(* Logix 5000 project; controller BTS01 vendor 1 type 14 code 217 rev 32.14; software revision 32.04; part 2 of 15 *)
(* tags used below, declared in another part *)
   V1101 : DTE_Air_Valve_v2;   // Tank 1100 Fill Valve
   V1102 : DTE_Air_Valve_v2;   // Tank 1100 Discharge Valve
   V1103 : DTE_Air_Valve_v2;   // Tank 1100 Line Valve
   V1201 : DTE_Air_Valve_v2;   // Tank 1200 Fill Valve
   V1202 : DTE_Air_Valve_v2;   // Tank 1200 Discharge Valve
   V1203 : DTE_Air_Valve_v2;   // Tank 1200 Line Valve

ADD_ON_INSTRUCTION SCP   (* revision 1.2, vendor Rockwell Automation *)
// Scale w/Parameters
// Help:
// Use this instruction to scale data from your analog module and bring it into the limits prescribed by the process variable or another analog module.
// Equations used in calculating a linear relationship:
// Scaled value = (input value - input min.) x rate + scaled minimum
// Rate = (scaled max. - scaled min.) / (input max. - input min.)
// Enabling the Limit_En Bit Limits the Output Value to the Scaled Min/Max Values. (09/16/16) DTK
VAR_INPUT
   Input : REAL; {required}
   Input_Min : REAL; {required}
   Input_Max : REAL; {required}
   Scaled_Min : REAL; {required}
   Scaled_Max : REAL; {required}
END_VAR
VAR_OUTPUT
   Output : REAL; {access Read Only, required}
END_VAR
VAR_INPUT
   Limit_En : BOOL; {visible}   // Limit Enable Bit Limits Output to Scaled Min/Max Values
END_VAR
VAR
   Rate : REAL;
END_VAR

ROUTINE Logic   (* ladder *)
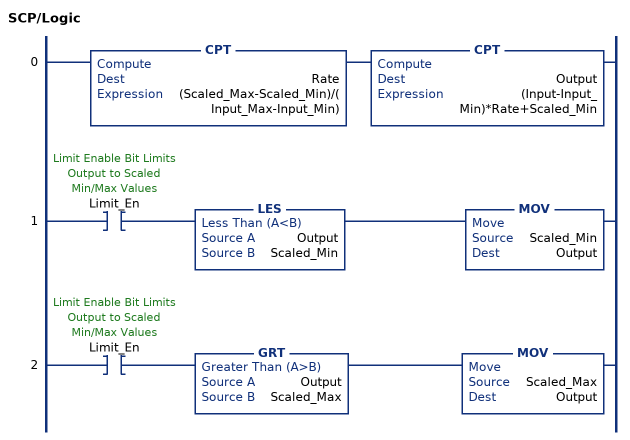
   0: CPT(Rate,(Scaled_Max-Scaled_Min)/(Input_Max-Input_Min))CPT(Output,(Input-Input_Min)*Rate+Scaled_Min);
   1: XIC(Limit_En)LES(Output,Scaled_Min)MOV(Scaled_Min,Output);
   2: XIC(Limit_En)GRT(Output,Scaled_Max)MOV(Scaled_Max,Output);
END_ROUTINE
END_ADD_ON_INSTRUCTION

ADD_ON_INSTRUCTION Temperature_Transmitter   (* revision 1.0 *)
VAR_INPUT
   RawInput : REAL; {required}   // Raw Input from Analog Input Card
   Input_Min : REAL; {required}   // I/O Module Scaling (MIN)
   Input_Max : REAL; {required}   // I/O Module Scaling (MAX)
   ScaledMin : REAL; {required}   // R/I Scaling (MIN)
   ScaledMax : REAL; {required}   // R/I Scaling (MAX)
   CalOffset : REAL; {required}   // Calibration Offset
END_VAR
VAR_OUTPUT
   MeasuredDegC : REAL; {access Read Only, visible}   // Sensor Temperature in Degrees C
   DegC : REAL; {access Read Only, visible}   // Display Temperature in Degrees C
   DegF : REAL; {access Read Only, visible}   // Display Temperature in Degrees F
END_VAR
VAR
   Offset : REAL;   // Linearity Offset
   Slope : REAL;   // Linearity Slope
END_VAR

ROUTINE Logic   (* ladder *)
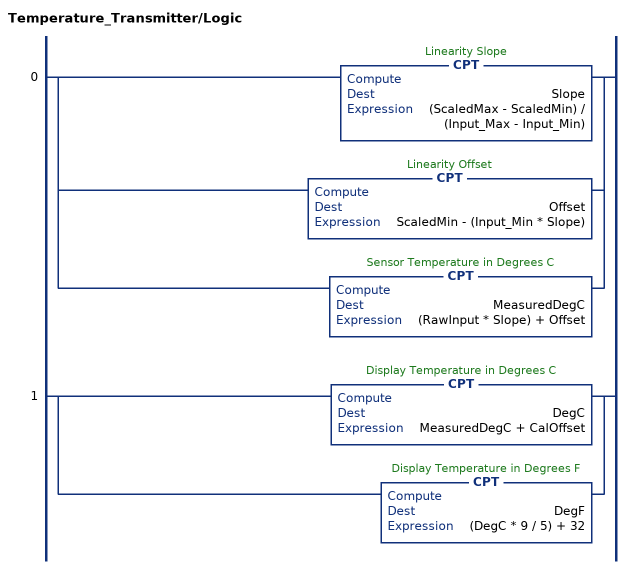
   0: [CPT(Slope,(ScaledMax - ScaledMin) / (Input_Max - Input_Min)) ,CPT(Offset,ScaledMin - (Input_Min * Slope)) ,CPT(MeasuredDegC,(RawInput * Slope) + Offset) ];
   1: [CPT(DegC,MeasuredDegC + CalOffset) ,CPT(DegF,(DegC * 9 / 5) + 32) ];
END_ROUTINE
END_ADD_ON_INSTRUCTION

ADD_ON_INSTRUCTION Toggle_Bit   (* revision 1.0 Created 4/01/2022 Sean Daehn *)
// Toggle Bit on and off with single momentary pushbutton
VAR_INPUT
   Toggle_PB : BOOL; {access None, required}
END_VAR
VAR_OUTPUT
   Output : BOOL; {access None, required}
END_VAR
VAR
   oneshot : BOOL; {access None}
   Toggle_On : BOOL; {access None}
   Toggle_Off : BOOL; {access None}
END_VAR

ROUTINE Logic   (* ladder *)
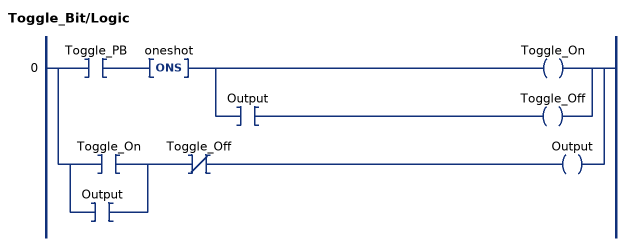
   0: [XIC(Toggle_PB) ONS(oneshot) [OTE(Toggle_On) ,XIC(Output) OTE(Toggle_Off) ] ,[XIC(Toggle_On) ,XIC(Output) ] XIO(Toggle_Off) OTE(Output) ];
END_ROUTINE
END_ADD_ON_INSTRUCTION

VAR_GLOBAL   (* controller tags *)
   ActiveRecipePF1000Interlock : DINT;
   AG1101 : DTE_VFD := (INTERLOCK := 1, SPEED_FWD := 20.0, AUTO_SPEED_SETPOINT := 20.0, FORCE_SPEED_SETPOINT := 10.0, ITEMTAG := 1101, MOA_MODE := 1);   // Tank 1100 Agitator
   AG1101_CIP_ENABLE : BOOL;
   AG1101_ONS : DINT := 1;
   AG1201 : DTE_VFD := (INTERLOCK := 1, SPEED_FWD := 20.0, AUTO_SPEED_SETPOINT := 20.0, FORCE_SPEED_SETPOINT := 20.0, ITEMTAG := 1201, MOA_MODE := 1);   // Tank 1200 Agitator
   AG1201_CIP_ENABLE : BOOL;
   AG1201_ONS : DINT;
   AirBlow_ONS : DINT;
   AirBlow_Timer : TIMER := (PRE := 30000);
   AirblowPB : BOOL;
   Alarm_Active : DINT;
   Alarm_TMR : TIMER[17,32] := ([0,0].PRE := 500, [0,1].PRE := 500, [0,2].PRE := 500, [0,3].PRE := 500, [0,4].PRE := 500, [0,5].PRE := 500, [0,6].PRE := 500, [0,7].PRE := 500, [0,8].PRE := 500, [0,9].PRE := 500, [0,10].PRE := 500, [0,11].PRE := 500, [0,12].PRE := 500, [0,13].PRE := 500, [0,14].PRE := 500, [0,15].PRE := 500, [0,16].PRE := 500, [0,17].PRE := 500, [0,18].PRE := 500, [0,19].PRE := 500, [0,20].PRE := 500, [0,21].PRE := 100, [0,22].PRE := 100, [0,23].PRE := 5000, [0,24].PRE := 5000, [0,25].PRE := 5000, [0,26].PRE := 5000, [0,27].PRE := 5000, [0,28].PRE := 5000, [0,29].PRE := 5000, [0,30].PRE := 5000, [0,31].PRE := 5000, [1,0].PRE := 100, [1,1].PRE := 100, [1,2].PRE := 500, [1,3].PRE := 500, [1,4].PRE := 500, [1,5].PRE := 500, [1,6].PRE := 500, [1,7].PRE := 500, [1,8].PRE := 2000, [1,9].PRE := 2000, [1,10].PRE := 2000, [1,11].PRE := 30000, [1,12].PRE := 5000, [1,13].PRE := 1000, [1,14].PRE := 10000, [1,15].PRE := 10000, [1,16].PRE := 10000, [1,18].PRE := 10000, [1,19].PRE := 10000, [1,20].PRE := 10000, [1,21].PRE := 10000, [1,22].PRE := 10000, [1,23].PRE := 10000, [1,24].PRE := 5000, [1,25].PRE := 1000, [2,0].PRE := 5000, [2,1].PRE := 5000, [2,2].PRE := 5000,
        [2,3].PRE := 5000, [2,4].PRE := 5000, [2,5].PRE := 5000, [2,6].PRE := 5000, [2,7].PRE := 5000, [2,8].PRE := 5000, [2,9].PRE := 5000, [2,10].PRE := 5000, [2,11].PRE := 5000, [2,12].PRE := 5000, [2,13].PRE := 5000, [2,14].PRE := 5000, [2,15].PRE := 5000, [2,16].PRE := 5000, [2,17].PRE := 5000, [2,18].PRE := 5000, [2,19].PRE := 5000, [2,20].PRE := 5000, [2,21].PRE := 5000, [2,22].PRE := 5000, [2,23].PRE := 5000, [2,24].PRE := 5000, [2,25].PRE := 5000, [2,26].PRE := 5000, [2,27].PRE := 5000, [2,28].PRE := 5000, [2,29].PRE := 5000, [2,30].PRE := 5000, [2,31].PRE := 5000, [3,4].PRE := 10000, [3,5].PRE := 10000, [3,6].PRE := 10000, [3,7].PRE := 10000, [3,8].PRE := 10000, [3,9].PRE := 10000, [3,10].PRE := 10000, [3,12].PRE := 10000, [3,13].PRE := 10000, [3,14].PRE := 500, [3,15].PRE := 60000, [3,16].PRE := 20000, [4,1].PRE := 10000, [4,2].PRE := 10000, [4,3].PRE := 10000, [4,4].PRE := 10000, [4,5].PRE := 10000, [4,6].PRE := 10000, [4,7].PRE := 10000, [4,8].PRE := 10000, [4,9].PRE := 10000, [4,10].PRE := 10000, [4,11].PRE := 10000, [4,12].PRE := 10000, [4,13].PRE := 10000, [4,14].PRE := 10000, [4,18].PRE := 5000, [4,19].PRE := 5000, [5,0].PRE := 10000, [5,1].PRE := 10000, [5,2].PRE := 10000,
        [5,3].PRE := 10000, [5,4].PRE := 10000, [5,5].PRE := 10000, [5,6].PRE := 10000, [5,7].PRE := 10000, [5,8].PRE := 10000, [5,9].PRE := 10000, [5,10].PRE := 10000, [5,11].PRE := 10000, [5,12].PRE := 10000, [5,13].PRE := 10000, [5,14].PRE := 10000, [5,15].PRE := 5000, [5,16].PRE := 5000, [6,0].PRE := 10000, [6,1].PRE := 10000, [6,2].PRE := 10000, [6,3].PRE := 10000, [6,4].PRE := 10000, [6,5].PRE := 10000, [6,6].PRE := 10000, [6,7].PRE := 10000, [6,8].PRE := 10000, [6,9].PRE := 10000, [6,10].PRE := 10000, [6,11].PRE := 10000, [6,12].PRE := 10000, [6,13].PRE := 10000, [6,14].PRE := 10000, [6,15].PRE := 5000, [6,16].PRE := 5000, [6,17].PRE := 5000, [7,0].PRE := 10000, [7,1].PRE := 10000, [7,2].PRE := 10000, [7,3].PRE := 10000, [7,4].PRE := 10000, [7,5].PRE := 10000, [7,6].PRE := 10000, [7,7].PRE := 10000, [7,8].PRE := 10000, [7,9].PRE := 10000, [7,10].PRE := 10000, [7,11].PRE := 10000, [7,12].PRE := 10000, [7,13].PRE := 10000, [7,14].PRE := 10000, [7,15].PRE := 5000, [7,16].PRE := 5000, [8,0].PRE := 10000, [8,1].PRE := 10000, [8,2].PRE := 10000, [8,3].PRE := 10000, [8,4].PRE := 10000, [8,5].PRE := 10000, [8,6].PRE := 10000, [8,7].PRE := 10000, [8,8].PRE := 10000, [8,9].PRE := 10000, [8,10].PRE := 10000,
        [8,11].PRE := 10000, [8,12].PRE := 10000, [8,13].PRE := 10000, [8,14].PRE := 10000, [8,15].PRE := 10000, [8,16].PRE := 10000, [8,17].PRE := 10000, [8,18].PRE := 10000, [8,19].PRE := 10000, [8,20].PRE := 10000, [8,21].PRE := 10000, [8,22].PRE := 10000, [8,23].PRE := 10000, [8,24].PRE := 10000, [8,25].PRE := 10000, [8,26].PRE := 10000, [8,27].PRE := 10000, [8,28].PRE := 10000, [8,29].PRE := 10000, [8,30].PRE := 2000, [8,31].PRE := 5000, [9,0].PRE := 5000, [9,1].PRE := 20000, [10,0].PRE := 10000, [10,1].PRE := 10000, [10,2].PRE := 10000, [10,3].PRE := 10000, [10,4].PRE := 10000, [10,5].PRE := 10000, [10,6].PRE := 10000, [10,7].PRE := 10000, [10,8].PRE := 10000, [10,9].PRE := 10000, [10,10].PRE := 20000, [11,0].PRE := 10000, [11,1].PRE := 10000, [11,2].PRE := 10000, [11,3].PRE := 10000, [11,4].PRE := 10000, [11,5].PRE := 10000, [11,6].PRE := 10000, [11,7].PRE := 10000, [11,8].PRE := 20000, [12,0].PRE := 10000, [12,1].PRE := 10000, [12,2].PRE := 10000, [12,3].PRE := 10000, [12,4].PRE := 10000, [12,5].PRE := 10000, [12,6].PRE := 10000, [12,7].PRE := 10000, [12,8].PRE := 10000, [12,9].PRE := 10000, [12,10].PRE := 10000, [12,11].PRE := 10000, [12,12].PRE := 20000, [14,0].PRE := 10000, [14,1].PRE := 10000, [14,2].PRE := 10000, [14,3].PRE := 10000,
        [14,4].PRE := 10000, [14,5].PRE := 10000, [14,6].PRE := 10000, [14,7].PRE := 10000, [14,8].PRE := 10000, [14,10].PRE := 10000, [14,11].PRE := 10000, [14,14].PRE := 10000, [14,15].PRE := 10000, [14,16].PRE := 10000, [14,17].PRE := 20000, [14,19].PRE := 20000, [14,20].PRE := 20000, [14,21].PRE := 20000, [14,22].PRE := 20000);
   ALM_ENABLE : DINT[25] := ([0] := 262143, [1] := 255);
   ApplyDST : SINT;
   C02S01 : REAL[8] := ([1] := 0.5937958);   // 5069-IF8
        [0]   // Tank 1100 Level Transmitter LT1101
        [1]   // Tank 1200 Level Transmitter LT1201
   C02S02 : REAL[8] := ([6] := 0.60912704);   // 5069-OF8
        [0]   // Tank 1100 Agitator Speed Ref VFD1101
        [1]   // Tank 1200 Agitator Speed Ref VFD1201
        [2]   // Bowl Chopper Disc Speed Reference VFD1001
        [3]   // Dressing Tank Disc Speed Reference VFD1002
        [4]   // CIP Return Pump Speed Reference VFD1003
        [5]   // Tank 1100 Remote Display
        [6]   // Tank 1200 Remote Display
   C02S03 : INT := 18773;   // 5069-IB16
        .0   // Emergency Stop Relay State
        .1   // Tank 1100 Agitator Run Signal VFD1101
        .10   // Filler Call for Product Signal
        .11   // CIP Cart Communications Connected
        .12   // P1001 Start Pushbutton
        .13   // P1001 Stop Pushbutton
        .14   // Filler CIP Return Pump Fault Signal VFD1004
        .15   // Filler CIP Return Pump Run Signal VFD1004
        .2   // Tank 1100 Agitator Fault Signal VFD1101
        .3   // Tank 1200 Agitator Run Signal VFD1201
        .4   // Tank 1200 Agitator Fault Signal VFD1201
        .5   // Bowl Chopper Disc Run Signal VFD1001
        .6   // Bowl Chopper Disc Fault Signal VFD1001
        .7   // Dressing Tank Disc Run Signal VFD1002
        .8   // CIP Return Pump Fault Signal VFD1003
        .9   // CIP Return Pump Run Signal VFD1003
   C02S04 : INT := 2;   // 5069-OB16
        .0   // V1001 Air Blow
        .1   // V1101
        .10   // V1005
        .11   // V1006
        .12   // V1007
        .2   // V1102
        .3   // V1103
        .4   // V1201
        .5   // V1202
        .6   // V1203
        .7   // V1002
        .8   // V1003
        .9   // V1004
   C02S05 : INT;   // 5069-OB16
        .0   // Tank 1100 Agitator Run Enable VFD1101
        .1   // Tank 1200 Agitator Run Enable VFD1201
        .2   // Bowl Chopper Disc Run Enable VFD1001
        .3   // Dressing Tank Disc Run Enable VFD1002
        .4   // CIP Return Pump Run Enable VFD1003
        .5   // CIP Cart Run Enable
        .6   // CIP Signal to Filler
        .7   // Filler CIP Return Pump Run Enable VFD1004
   C02S06 : INT := -28656;   // 5069-IB16
        .0   // Flow Switch FS1
        .1   // Prox Switch ZS1000-1
        .10   // Prox Switch ZS1001-3 (Future)
        .11   // Prox Switch ZS1001-4
        .12   // Prox Switch ZS1001-5
        .15   // Dressing Tank Disc Fault Signal VFD1002
        .2   // Prox Switch ZS1000-2
        .3   // Prox Switch ZS1000-3
        .4   // Prox Switch ZS1000-4
        .5   // Prox Switch ZS1000-5 (Future)
        .6   // Prox Switch ZS1101
        .7   // Prox Switch ZS1201
        .8   // Prox Switch ZS1001-1
        .9   // Prox Switch ZS1001-2 (Future)
   CAUSTIC1_TIME_REM : DINT;   // CIP 1 CAUSTIC TIM REMAINING
   CAUSTIC_DRAIN_LATCH : BOOL;
   CAUSTIC_DRAIN_RUN : BOOL;
   CAUSTIC_DRAIN_RUN_CLR : BOOL;
   CAUSTIC_DRAIN_RUN_PB : BOOL;
   Caustic_Fill_Latch : BOOL;   // Caustic Tank Fill Latch
   CAUSTIC_FILL_PB_HMI : BOOL;
   CAUSTIC_FILL_RUN : BOOL;
   CAUSTIC_FILL_RUN_CLR : BOOL;
   CAUSTIC_PREP_LATCH : BOOL;
   CAUSTIC_PREP_RUN : BOOL;
   CAUSTIC_PREP_RUN_CLR : BOOL;   // CAUSTIC PREP JKFF CLEAR BIT
   CAUSTIC_PREP_RUN_PB : BOOL;
   CAUSTIC_PREP_TEMP_SPT : REAL := 145.0;
   CAUSTIC_PREP_TIME_SPT : REAL := 10.0;
   CAUSTIC_TANK_LEVEL_OFF_PERC : DINT := 100;   // HMI INPUT OF WATER LEVEL OFF IN %
   CIP1_CAUSTIC_DRAIN_FILE : DINT := 268435466;   // CIP 1 RAW RECIEVING CIP CAUSTIC DRAIN ENABLE REFERENCE FILE
   CIP1_CAUSTIC_PREP_FILE : DINT := 304611370;   // CIP 1 RAW RECIEVING CIP CAUSTIC PREP ENABLE REFERENCE FILE
   CIP1_FINALRINSE_DRAIN_FILE : DINT := 268435978;   // CIP 1 RAW RECIEVING CIP FINAL RINSE DRAIN ENABLE REFERENCE FILE
   CIP1_PRERINSE_DRAIN_FILE : DINT := 268435465;   // CIP 1 RAW RECIEVING CIP PRERINSE DRAIN ENABLE REFERENCE FILE
   CIP1_PRERINSE_PREP_FILE : DINT := 285474889;   // CIP 1 RAW RECIEVING CIP PRERINSE PREP ENABLE REFERENCE FILE
   CIP1_SUPPLY_TEMP_OFFSET : DINT;   // CIP 1 SUPPLY TEMP OFFSET FROM RETURN TEMP SETPOINT
   CIP_1_ACTIVE_CIRCUIT : DINT;
   CIP_1_ACTIVE_PROGRAM : CIP_PROGRAM := (STEPS[0].NAME := 'NOT IN USE', STEPS[1].TYPE := 999, STEPS[2].TYPE := 999, STEPS[3].TYPE := 999, STEPS[4].TYPE := 999, STEPS[5].TYPE := 999, STEPS[6].TYPE := 999, STEPS[7].TYPE := 999, STEPS[8].TYPE := 999, STEPS[9].TYPE := 999, STEPS[10].TYPE := 999, STEPS[11].TYPE := 999, STEPS[12].TYPE := 999, STEPS[13].TYPE := 999, STEPS[14].TYPE := 999, STEPS[15].TYPE := 999, STEPS[16].TYPE := 999, STEPS[17].TYPE := 999, STEPS[18].TYPE := 999, STEPS[19].TYPE := 999, STEPS[20].TYPE := 999, STEPS[21].TYPE := 999, STEPS[22].TYPE := 999, STEPS[23].TYPE := 999, STEPS[24].TYPE := 999, STEPS[25].TYPE := 999, STEPS[26].TYPE := 999, STEPS[27].TYPE := 999, STEPS[28].TYPE := 999, STEPS[29].TYPE := 999, STEPS[30].TYPE := 999, STEPS[31].TYPE := 999, STEPS[32].TYPE := 999, STEPS[33].TYPE := 999, STEPS[34].TYPE := 999, STEPS[35].TYPE := 999, STEPS[36].TYPE := 999, STEPS[37].TYPE := 999, STEPS[38].TYPE := 999, STEPS[39].TYPE := 999, STEPS[40].TYPE := 999, STEPS[41].TYPE := 999, STEPS[42].TYPE := 999, STEPS[43].TYPE := 999, STEPS[44].TYPE := 999, STEPS[45].TYPE := 999, STEPS[46].TYPE := 999, STEPS[47].TYPE := 999, STEPS[48].TYPE := 999, STEPS[49].TYPE := 999);
   CIP_1_ACTIVE_PROGRAM_SPANISH : CIP_PROGRAM;
   CIP_1_ACTIVE_STEP : CIP_STEP_DEF := (NAME := 'NOT IN USE');   // CIP 1 ACTIVE STEP DATA
   CIP_1_ACTIVE_STEP_NUMBER : DINT;
   CIP_1_ACTIVE_STEP_SUP_TEMP : DINT;   // CIP 1 SUPPLY TEMP SETPOINT FOR ACTIVE STEP
   CIP_1_ACTIVE_STEP_TIME : DINT;
   CIP_1_ALARM_INDICATOR : DINT;   // ALARM STATE INDICATOR AT HMI
   CIP_1_ALARMS : DINT[30];
   CIP_1_AVAIL_STEP_ID : DINT := 1;
   CIP_1_CAUSTIC_TRANS_ACT : BOOL;   // CIP 1 RETURN TO CAUSTIC TANK LEVEL TRANSITION ACTIVE
   CIP_1_Circuit1_Prox_Mismatch : BOOL;
   CIP_1_Circuit1_Tank_Not_Empty : BOOL;
   CIP_1_Circuit2_Prox_Mismatch : BOOL;
   CIP_1_Circuit2_Tank_Not_Empty : BOOL;
   CIP_1_Circuit3_Prox_Mismatch : BOOL;
   CIP_1_Circuit4_Prox_Mismatch : BOOL;
   CIP_1_CIRCUIT_SELECT_EDIT_HMI : INT := 1;
   CIP_1_CIRCUIT_SELECT_EDIT_HMI_NAME : STRING[50];
   CIP_1_CIRCUIT_SELECT_HMI : INT := 4;
   CIP_1_CURRENT_STEP_MESSAGE_INT : DINT := -1;
   CIP_1_EDIT_PROGRAM : CIP_PROGRAM := (NAME := 'Dressing Tank 1100 Wash', NUMBER := 1, STEPS[0].NAME := 'SYSTEM IDLE', STEPS[1].NAME := 'OPERATOR ACKNOWLEDGE', STEPS[1].TYPE := 50, STEPS[2].NAME := 'PRERINSE', STEPS[2].TYPE := 100, STEPS[2].TIME_SPT := 5.0, STEPS[2].REF_FILE := 5125, STEPS[3].NAME := 'PRERINSE PUMP DOWN', STEPS[3].TYPE := 400, STEPS[3].TIME_SPT := 0.5, STEPS[3].REF_FILE := 4101, STEPS[4].NAME := 'CAUSTIC WASH (TIME ONLY)', STEPS[4].TYPE := 300, STEPS[4].TIME_SPT := 30.0, STEPS[4].REF_FILE := 5125, STEPS[5].NAME := 'CAUSTIC PUMP DOWN', STEPS[5].TYPE := 400, STEPS[5].TIME_SPT := 0.5, STEPS[5].REF_FILE := 4101, STEPS[6].NAME := 'POST RINSE', STEPS[6].TYPE := 100, STEPS[6].TIME_SPT := 5.0, STEPS[6].REF_FILE := 5125, STEPS[7].NAME := 'SANITIZER', STEPS[7].TYPE := 600, STEPS[7].TIME_SPT := 5.0, STEPS[7].REF_FILE := 5125, STEPS[8].NAME := 'SANITIZER PUMP DOWN', STEPS[8].TYPE := 400, STEPS[8].TIME_SPT := 0.5, STEPS[8].REF_FILE := 4101, STEPS[9].NAME := 'FINAL RINSE TO DRAIN', STEPS[9].TYPE := 100, STEPS[9].TIME_SPT := 5.0, STEPS[9].REF_FILE := 5125, STEPS[10].NAME := 'FINAL RINSE PUMP DOWN', STEPS[10].TYPE := 400, STEPS[10].TIME_SPT := 0.5, STEPS[10].REF_FILE := 4101, STEPS[11].TYPE := 999, STEPS[12].TYPE := 999, STEPS[13].TYPE := 999, STEPS[14].TYPE := 999, STEPS[15].TYPE := 999, STEPS[16].TYPE := 999, STEPS[17].TYPE := 999, STEPS[18].TYPE := 999, STEPS[19].TYPE := 999, STEPS[20].TYPE := 999, STEPS[21].TYPE := 999, STEPS[22].TYPE := 999, STEPS[23].TYPE := 999, STEPS[24].TYPE := 999, STEPS[25].TYPE := 999, STEPS[26].TYPE := 999, STEPS[27].TYPE := 999, STEPS[28].TYPE := 999, STEPS[29].TYPE := 999,
        STEPS[30].TYPE := 999, STEPS[31].TYPE := 999, STEPS[32].TYPE := 999, STEPS[33].TYPE := 999, STEPS[34].TYPE := 999, STEPS[35].TYPE := 999, STEPS[36].TYPE := 999, STEPS[37].TYPE := 999, STEPS[38].TYPE := 999, STEPS[39].TYPE := 999, STEPS[40].TYPE := 999, STEPS[41].TYPE := 999, STEPS[42].TYPE := 999, STEPS[43].TYPE := 999, STEPS[44].TYPE := 999, STEPS[45].TYPE := 999, STEPS[46].TYPE := 999, STEPS[47].TYPE := 999, STEPS[48].TYPE := 999, STEPS[49].TYPE := 999);
   CIP_1_FLOW_PROOF : BOOL;   // CIP 1 FLOW PROOF BIT 0 = NO FLOW 1 = FLOW
   CIP_1_HOLD_LATCH : BOOL;
   CIP_1_HOLD_PB_CTU : COUNTER;
   CIP_1_HOLD_PB_HMI : BOOL;
   CIP_1_HOLD_TIME : REAL;
   CIP_1_INSERT_STEP : DINT := 1;   // CIP1 INSERT STEP POINTER
   CIP_1_LOAD_ACTIVE_CIP_RECIPE_PB : BOOL;
   CIP_1_LOAD_RECIPE_EDIT_PB : BOOL;
   CIP_1_MASTER_REF_FILE : DINT[15,30] := ([0,1] := 2#1000_0000_0001_1100_0000_0010_0001_1000, [0,2] := 2#1001_0001_0000_0100_0000_0011_1001_1001, [0,3] := 2#1001_0001_0000_0100_0000_0010_0001_1001, [0,4] := 2#1000_0000_0000_0100_0000_0010_0001_1000, [0,5] := 2#1001_0001_0000_0100_0000_0010_0101_1001, [0,6] := 2#1001_0001_0000_0100_0000_0010_0001_1001, [0,7] := 2#1000_0000_0000_0000_0000_0110_0001_0000, [0,8] := 2#1001_0010_0010_1000_0000_0000_0011_1010, [0,9] := 2#1001_0010_0010_1000_0000_0000_0011_1010, [0,10] := 2#1001_0010_0010_1000_0000_0000_0011_1010, [0,11] := 2#1000_0000_0000_0000_0000_0000_0011_1000, [0,12] := 2#1001_0000_0001_0000_0000_0000_0011_1100, [0,13] := 2#1000_0000_0001_0000_0000_0100_0101_0000, [0,14] := 2#1000_0000_0001_0000_0000_0000_0101_1000, [0,15] := 2#1001_0000_0001_0000_0000_0000_0001_1100, [0,16] := 2#1001_0000_0001_0000_0000_0000_0001_1100, [0,17] := 2#1001_0000_1001_0000_0000_0000_0001_1100, [0,18] := 2#1001_0000_1001_0000_0000_0000_0001_1100, [0,19] := 2#1000_0000_0001_0000_0000_0100_0001_0000, [0,20] := 2#1000_0000_0001_0000_0000_0000_0001_1000, [0,21] := 2#0000_0000_0000_0000_0000_0000_0001_1000, [1,1] := 2#1000_0000_0001_1100_1000_1010_0001_1000, [1,2] := 2#1001_0001_0000_0100_1000_1010_0001_1001, [1,3] := 2#1001_0001_0000_0100_1000_1010_0001_1001, [1,4] := 2#1000_0000_0000_0100_1000_1010_0001_1000, [1,5] := 2#1001_0001_0000_0100_1000_1010_0101_1001, [1,6] := 2#1001_0001_0000_0100_1000_1010_0001_1001, [1,7] := 2#1000_0000_0000_0000_1000_1110_0001_0000, [1,8] := 2#1001_0010_0010_1000_1000_1000_0011_1010, [1,9] := 2#1001_0010_0010_1000_1000_1000_0011_1010, [1,10] := 2#1001_0010_0010_1000_1000_1000_0011_1010, [1,11] := 2#1000_0000_0000_0000_1000_1000_0011_1000, [1,12] := 2#1001_0000_0001_0000_1000_1000_0011_1100, [1,13] := 2#1000_0000_0001_0000_1000_1100_0101_0100, [1,14] := 2#1000_0000_0001_0000_1000_1000_0101_1000, [1,15] := 2#1001_0000_0001_0000_1000_1000_0001_1100, [1,16] := 2#1001_0000_0001_0000_1000_1000_0001_1100, [1,17] := 2#1001_0000_1001_0000_1000_1000_0001_1100, [1,18] := 2#1001_0000_1001_0000_1000_1000_0001_1100, [1,19] := 2#1000_0000_0001_0000_1000_1100_0001_0000, [1,20] := 2#1000_0000_0001_0000_1000_1000_0001_1000, [1,21] := 2#0000_0000_0000_0000_1000_1000_0001_1000, [3,1] := 2#1000_0000_0001_1100_0001_0010_0001_1000, [3,2] := 2#1001_0001_0000_0100_0001_0010_0001_1001, [3,3] := 2#1001_0001_0000_0100_0001_0010_0001_1001, [3,4] := 2#1000_0000_0000_0100_0001_0010_0001_1000, [3,5] := 2#1001_0001_0000_0100_0001_0010_0101_1001, [3,6] := 2#1001_0001_0000_0100_0001_0010_0001_1001, [3,7] := 2#1000_0000_0000_0000_0001_0110_0001_0000, [3,8] := 2#1001_0010_0010_1000_0001_0000_0011_1010, [3,9] := 2#1001_0010_0010_1000_0001_0000_0011_1010, [3,10] := 2#1001_0010_0010_1000_0001_0000_0011_1010, [3,11] := 2#1000_0000_0000_0000_0001_0000_0011_1000, [3,12] := 2#1001_0000_0001_0000_0001_0000_0011_1100, [3,13] := 2#1000_0000_0001_0000_0001_0100_0101_0100, [3,14] := 2#1000_0000_0001_0000_0001_0000_0101_1000, [3,15] := 2#1001_0000_0001_0000_0001_0000_0001_1100, [3,16] := 2#1001_0000_0001_0000_0001_0000_0001_1100, [3,17] := 2#1001_0000_1001_0000_0001_0000_0001_1100, [3,18] := 2#1001_0000_1001_0000_0001_0000_0001_1100,
        [3,19] := 2#1000_0000_0001_0000_0001_0100_0001_0000, [3,20] := 2#1000_0000_0001_0000_0001_0000_0001_1000, [3,21] := 2#0000_0000_0000_0000_0001_0000_0001_1000, [5,1] := 2#1000_0000_0001_1100_0100_1010_0001_1000, [5,2] := 2#1001_0001_0000_0100_0100_1010_0001_1001, [5,3] := 2#1001_0001_0000_0100_0100_1010_0001_1001, [5,4] := 2#1000_0000_0000_0100_0100_1010_0001_1000, [5,5] := 2#1001_0001_0000_0100_0100_1010_0101_1001, [5,6] := 2#1001_0001_0000_0100_0100_1010_0001_1001, [5,7] := 2#1000_0000_0000_0000_0100_1110_0001_0000, [5,8] := 2#1001_0010_0010_1000_0100_1000_0011_1010, [5,9] := 2#1001_0010_0010_1000_0100_1000_0011_1010, [5,10] := 2#1001_0010_0010_1000_0100_1000_0011_1010, [5,11] := 2#1000_0000_0000_0000_0100_1000_0011_1000, [5,12] := 2#1001_0000_0001_0000_0100_1000_0011_1100, [5,13] := 2#1000_0000_0001_0000_0100_1100_0101_0100, [5,14] := 2#1000_0000_0001_0000_0100_1000_0101_1000, [5,15] := 2#1001_0000_0001_0000_0100_1000_0001_1100, [5,16] := 2#1001_0000_0001_0000_0100_1000_0001_1100, [5,17] := 2#1001_0000_1001_0000_0100_1000_0001_1100, [5,18] := 2#1001_0000_1001_0000_0100_1000_0001_1100, [5,19] := 2#1000_0000_0001_0000_0100_1100_0001_0000, [5,20] := 2#1000_0000_0001_0000_0100_1000_0001_1000, [5,21] := 2#0000_0000_0000_0000_0100_1000_0001_1000, [7,1] := 2#1000_0000_0001_1100_0010_0010_0001_1000, [7,2] := 2#1001_0001_0000_0100_0010_0010_0001_1001, [7,3] := 2#1001_0001_0000_0100_0010_0010_0001_1001, [7,4] := 2#1000_0000_0000_0100_0010_0010_0001_1000, [7,5] := 2#1001_0001_0000_0100_0010_0010_0101_1001, [7,6] := 2#1001_0001_0000_0100_0010_0010_0001_1001, [7,7] := 2#1000_0000_0000_0000_0010_0110_0001_0000, [7,8] := 2#1001_0010_0010_1000_0010_0000_0011_1010, [7,9] := 2#1001_0010_0010_1000_0010_0000_0011_1010, [7,10] := 2#1001_0010_0010_1000_0010_0000_0011_1010, [7,11] := 2#1000_0000_0000_0000_0010_0000_0011_1000, [7,12] := 2#1001_0000_0001_0000_0010_0000_0011_1100, [7,13] := 2#1000_0000_0001_0000_0010_0100_0101_0100, [7,14] := 2#1000_0000_0001_0000_0010_0000_0101_1000, [7,15] := 2#1001_0000_0001_0000_0010_0000_0001_1100, [7,16] := 2#1001_0000_0001_0000_0010_0000_0001_1100, [7,17] := 2#1001_0000_1001_0000_0010_0000_0001_1100, [7,18] := 2#1001_0000_1001_0000_0010_0000_0001_1100, [7,19] := 2#1000_0000_0001_0000_0010_0100_0001_0000, [7,20] := 2#1000_0000_0001_0000_0010_0000_0001_1000, [7,21] := 2#0000_0000_0000_0000_0010_0000_0001_1000, [9,1] := 2#1000_0000_0001_1100_1100_1010_0001_1000, [9,2] := 2#1001_0001_0000_0100_1100_1010_0001_1001, [9,3] := 2#1001_0001_0000_0100_1100_1010_0001_1001, [9,4] := 2#1000_0000_0000_0100_1100_1010_0001_1000, [9,5] := 2#1001_0001_0000_0100_1100_1010_0101_1001, [9,6] := 2#1001_0001_0000_0100_1100_1010_0001_1001, [9,7] := 2#1000_0000_0000_0000_1100_1110_0001_0000, [9,8] := 2#1001_0010_0010_1000_1100_1000_0011_1010, [9,9] := 2#1001_0010_0010_1000_1100_1000_0011_1010, [9,10] := 2#1001_0010_0010_1000_1100_1000_0011_1010, [9,11] := 2#1000_0000_0000_0000_1100_1000_0011_1000, [9,12] := 2#1001_0000_0001_0000_1100_1000_0011_1100, [9,13] := 2#1000_0000_0001_0000_1100_1100_0101_0100, [9,14] := 2#1000_0000_0001_0000_1100_1000_0101_1000, [9,15] := 2#1001_0000_0001_0000_1100_1000_0001_1100,
        [9,16] := 2#1001_0000_0001_0000_1100_1000_0001_1100, [9,17] := 2#1001_0000_1001_0000_1100_1000_0001_1100, [9,18] := 2#1001_0000_1001_0000_1100_1000_0001_1100, [9,19] := 2#1000_0000_0001_0000_1100_1100_0001_0000, [9,20] := 2#1000_0000_0001_0000_1100_1000_0001_1000, [9,21] := 2#0000_0000_0000_0000_1100_1000_0001_1000, [11,1] := 2#1000_0000_0001_1100_0011_0010_0001_1000, [11,2] := 2#1001_0001_0000_0100_0011_0010_0001_1001, [11,3] := 2#1001_0001_0000_0100_0011_0010_0001_1001, [11,4] := 2#1000_0000_0000_0100_0011_0010_0001_1000, [11,5] := 2#1001_0001_0000_0100_0011_0010_0101_1001, [11,6] := 2#1001_0001_0000_0100_0011_0010_0001_1001, [11,7] := 2#1000_0000_0000_0000_0011_0110_0001_0000, [11,8] := 2#1001_0010_0010_1000_0011_0000_0011_1010, [11,9] := 2#1001_0010_0010_1000_0011_0000_0011_1010, [11,10] := 2#1001_0010_0010_1000_0011_0000_0011_1010, [11,11] := 2#1000_0000_0000_0000_0011_0000_0011_1000, [11,12] := 2#1001_0000_0001_0000_0011_0000_0011_1100, [11,13] := 2#1000_0000_0001_0000_0011_0100_0101_0100, [11,14] := 2#1000_0000_0001_0000_0011_0000_0101_1000, [11,15] := 2#1001_0000_0001_0000_0011_0000_0001_1100, [11,16] := 2#1001_0000_0001_0000_0011_0000_0001_1100, [11,17] := 2#1001_0000_1001_0000_0011_0000_0001_1100, [11,18] := 2#1001_0000_1001_0000_0011_0000_0001_1100, [11,19] := 2#1000_0000_0001_0000_0011_0100_0001_0000, [11,20] := 2#1000_0000_0001_0000_0011_0000_0001_1000, [11,21] := 2#0000_0000_0000_0000_0011_0000_0001_1000);   // SEQUENCER PINS CIP 1
   CIP_1_OPERATOR_ACK : BOOL;   // CIP 1 SEQUENCER OPERATOR ACKNOWLEDGE
   CIP_1_OPERATOR_ACK_PB_HMI : BOOL;
   CIP_1_PERMISSION : BOOL;
   CIP_1_PRERINSE_TRANS_ACT : BOOL;   // CIP 1 RETURN TO PRERINSE TANK LEVEL TRANSITION ACTIVE
   CIP_1_PRERINSE_TRANS_DRAIN : BOOL;   // CIP 1 RETURN TO PRERINSE TANK LEVEL TRANSITION ACTIVE
   CIP_1_PROGRAM_ID : INT := 1;
   CIP_1_PROGRAMS : CIP_PROGRAM[30] := ([0].STEPS[0].NAME := 'NOT IN USE', [0].STEPS[1].TYPE := 999, [0].STEPS[2].TYPE := 999, [0].STEPS[3].TYPE := 999, [0].STEPS[4].TYPE := 999, [0].STEPS[5].TYPE := 999, [0].STEPS[6].TYPE := 999, [0].STEPS[7].TYPE := 999, [0].STEPS[8].TYPE := 999, [0].STEPS[9].TYPE := 999, [0].STEPS[10].TYPE := 999, [0].STEPS[11].TYPE := 999, [0].STEPS[12].TYPE := 999, [0].STEPS[13].TYPE := 999, [0].STEPS[14].TYPE := 999, [0].STEPS[15].TYPE := 999, [0].STEPS[16].TYPE := 999, [0].STEPS[17].TYPE := 999, [0].STEPS[18].TYPE := 999, [0].STEPS[19].TYPE := 999, [0].STEPS[20].TYPE := 999, [0].STEPS[21].TYPE := 999, [0].STEPS[22].TYPE := 999, [0].STEPS[23].TYPE := 999, [0].STEPS[24].TYPE := 999, [0].STEPS[25].TYPE := 999, [0].STEPS[26].TYPE := 999, [0].STEPS[27].TYPE := 999, [0].STEPS[28].TYPE := 999, [0].STEPS[29].TYPE := 999, [0].STEPS[30].TYPE := 999, [0].STEPS[31].TYPE := 999, [0].STEPS[32].TYPE := 999, [0].STEPS[33].TYPE := 999, [0].STEPS[34].TYPE := 999, [0].STEPS[35].TYPE := 999, [0].STEPS[36].TYPE := 999, [0].STEPS[37].TYPE := 999, [0].STEPS[38].TYPE := 999, [0].STEPS[39].TYPE := 999, [0].STEPS[40].TYPE := 999, [0].STEPS[41].TYPE := 999, [0].STEPS[42].TYPE := 999, [0].STEPS[43].TYPE := 999, [0].STEPS[44].TYPE := 999, [0].STEPS[45].TYPE := 999, [0].STEPS[46].TYPE := 999, [0].STEPS[47].TYPE := 999, [0].STEPS[48].TYPE := 999, [0].STEPS[49].TYPE := 999, [1].NAME := 'Dressing Tank 1100 Wash', [1].NUMBER := 1, [1].STEPS[0].NAME := 'SYSTEM IDLE', [1].STEPS[1].NAME := 'OPERATOR ACKNOWLEDGE', [1].STEPS[1].TYPE := 50, [1].STEPS[2].NAME := 'PRERINSE', [1].STEPS[2].TYPE := 100, [1].STEPS[2].TIME_SPT := 5.0, [1].STEPS[2].REF_FILE := 5125, [1].STEPS[3].NAME := 'PRERINSE PUMP DOWN',
        [1].STEPS[3].TYPE := 400, [1].STEPS[3].TIME_SPT := 0.5, [1].STEPS[3].REF_FILE := 4101, [1].STEPS[4].NAME := 'CAUSTIC WASH (TIME ONLY)', [1].STEPS[4].TYPE := 300, [1].STEPS[4].TIME_SPT := 30.0, [1].STEPS[4].REF_FILE := 5125, [1].STEPS[5].NAME := 'CAUSTIC PUMP DOWN', [1].STEPS[5].TYPE := 400, [1].STEPS[5].TIME_SPT := 0.5, [1].STEPS[5].REF_FILE := 4101, [1].STEPS[6].NAME := 'POST RINSE', [1].STEPS[6].TYPE := 100, [1].STEPS[6].TIME_SPT := 5.0, [1].STEPS[6].REF_FILE := 5125, [1].STEPS[7].NAME := 'SANITIZER', [1].STEPS[7].TYPE := 600, [1].STEPS[7].TIME_SPT := 5.0, [1].STEPS[7].REF_FILE := 5125, [1].STEPS[8].NAME := 'SANITIZER PUMP DOWN', [1].STEPS[8].TYPE := 400, [1].STEPS[8].TIME_SPT := 0.5, [1].STEPS[8].REF_FILE := 4101, [1].STEPS[9].NAME := 'FINAL RINSE TO DRAIN', [1].STEPS[9].TYPE := 100, [1].STEPS[9].TIME_SPT := 5.0, [1].STEPS[9].REF_FILE := 5125, [1].STEPS[10].NAME := 'FINAL RINSE PUMP DOWN', [1].STEPS[10].TYPE := 400, [1].STEPS[10].TIME_SPT := 0.5, [1].STEPS[10].REF_FILE := 4101, [1].STEPS[11].TYPE := 999, [1].STEPS[12].TYPE := 999, [1].STEPS[13].TYPE := 999, [1].STEPS[14].TYPE := 999, [1].STEPS[15].TYPE := 999, [1].STEPS[16].TYPE := 999, [1].STEPS[17].TYPE := 999, [1].STEPS[18].TYPE := 999, [1].STEPS[19].TYPE := 999, [1].STEPS[20].TYPE := 999, [1].STEPS[21].TYPE := 999, [1].STEPS[22].TYPE := 999, [1].STEPS[23].TYPE := 999, [1].STEPS[24].TYPE := 999, [1].STEPS[25].TYPE := 999, [1].STEPS[26].TYPE := 999, [1].STEPS[27].TYPE := 999, [1].STEPS[28].TYPE := 999, [1].STEPS[29].TYPE := 999, [1].STEPS[30].TYPE := 999, [1].STEPS[31].TYPE := 999, [1].STEPS[32].TYPE := 999, [1].STEPS[33].TYPE := 999, [1].STEPS[34].TYPE := 999, [1].STEPS[35].TYPE := 999, [1].STEPS[36].TYPE := 999, [1].STEPS[37].TYPE := 999, [1].STEPS[38].TYPE := 999, [1].STEPS[39].TYPE := 999,
        [1].STEPS[40].TYPE := 999, [1].STEPS[41].TYPE := 999, [1].STEPS[42].TYPE := 999, [1].STEPS[43].TYPE := 999, [1].STEPS[44].TYPE := 999, [1].STEPS[45].TYPE := 999, [1].STEPS[46].TYPE := 999, [1].STEPS[47].TYPE := 999, [1].STEPS[48].TYPE := 999, [1].STEPS[49].TYPE := 999, [2].NAME := 'Dressing Tank 1200 Wash', [2].NUMBER := 2, [2].STEPS[0].NAME := 'SYSTEM IDLE', [2].STEPS[1].NAME := 'OPERATOR ACKNOWLEDGE', [2].STEPS[1].TYPE := 50, [2].STEPS[1].REF_FILE := 4, [2].STEPS[2].NAME := 'PRERINSE', [2].STEPS[2].TYPE := 100, [2].STEPS[2].TIME_SPT := 5.0, [2].STEPS[2].REF_FILE := 163845, [2].STEPS[3].NAME := 'PRERINSE PUMP DOWN', [2].STEPS[3].TYPE := 400, [2].STEPS[3].TIME_SPT := 0.5, [2].STEPS[3].REF_FILE := 131077, [2].STEPS[4].NAME := 'CAUSTIC WASH (TIME ONLY)', [2].STEPS[4].TYPE := 300, [2].STEPS[4].TIME_SPT := 30.0, [2].STEPS[4].REF_FILE := 163845, [2].STEPS[5].NAME := 'CAUSTIC PUMP DOWN', [2].STEPS[5].TYPE := 400, [2].STEPS[5].TIME_SPT := 0.5, [2].STEPS[5].REF_FILE := 131077, [2].STEPS[6].NAME := 'POST RINSE', [2].STEPS[6].TYPE := 100, [2].STEPS[6].TIME_SPT := 5.0, [2].STEPS[6].REF_FILE := 163845, [2].STEPS[7].NAME := 'SANITIZER', [2].STEPS[7].TYPE := 600, [2].STEPS[7].TIME_SPT := 5.0, [2].STEPS[7].REF_FILE := 131077, [2].STEPS[8].NAME := 'SANITIZER PUMP DOWN', [2].STEPS[8].TYPE := 400, [2].STEPS[8].TIME_SPT := 0.5, [2].STEPS[8].REF_FILE := 163845, [2].STEPS[9].NAME := 'FINAL RINSE TO DRAIN', [2].STEPS[9].TYPE := 100, [2].STEPS[9].TIME_SPT := 5.0, [2].STEPS[9].REF_FILE := 131077, [2].STEPS[10].NAME := 'FINAL RINSE PUMP DOWN', [2].STEPS[10].TYPE := 400, [2].STEPS[10].TIME_SPT := 0.5, [2].STEPS[10].REF_FILE := 131077, [2].STEPS[11].TYPE := 999, [2].STEPS[12].TYPE := 999, [2].STEPS[13].TYPE := 999, [2].STEPS[14].TYPE := 999, [2].STEPS[15].TYPE := 999, [2].STEPS[16].TYPE := 999, [2].STEPS[17].TYPE := 999, [2].STEPS[18].TYPE := 999,
        [2].STEPS[19].TYPE := 999, [2].STEPS[20].TYPE := 999, [2].STEPS[21].TYPE := 999, [2].STEPS[22].TYPE := 999, [2].STEPS[23].TYPE := 999, [2].STEPS[24].TYPE := 999, [2].STEPS[25].TYPE := 999, [2].STEPS[26].TYPE := 999, [2].STEPS[27].TYPE := 999, [2].STEPS[28].TYPE := 999, [2].STEPS[29].TYPE := 999, [2].STEPS[30].TYPE := 999, [2].STEPS[31].TYPE := 999, [2].STEPS[32].TYPE := 999, [2].STEPS[33].TYPE := 999, [2].STEPS[34].TYPE := 999, [2].STEPS[35].TYPE := 999, [2].STEPS[36].TYPE := 999, [2].STEPS[37].TYPE := 999, [2].STEPS[38].TYPE := 999, [2].STEPS[39].TYPE := 999, [2].STEPS[40].TYPE := 999, [2].STEPS[41].TYPE := 999, [2].STEPS[42].TYPE := 999, [2].STEPS[43].TYPE := 999, [2].STEPS[44].TYPE := 999, [2].STEPS[45].TYPE := 999, [2].STEPS[46].TYPE := 999, [2].STEPS[47].TYPE := 999, [2].STEPS[48].TYPE := 999, [2].STEPS[49].TYPE := 999, [3].NAME := 'Chopper Line Wash', [3].NUMBER := 3, [3].STEPS[0].NAME := 'SYSTEM IDLE', [3].STEPS[1].NAME := 'OPERATOR ACKNOWLEDGE', [3].STEPS[1].TYPE := 50, [3].STEPS[1].REF_FILE := 2097152, [3].STEPS[2].NAME := 'PRERINSE', [3].STEPS[2].TYPE := 100, [3].STEPS[2].TIME_SPT := 5.0, [3].STEPS[2].REF_FILE := 2164745, [3].STEPS[3].NAME := 'PRERINSE TO DRAIN', [3].STEPS[3].TYPE := 100, [3].STEPS[3].TIME_SPT := 0.5, [3].STEPS[3].REF_FILE := 2164745, [3].STEPS[4].NAME := 'CAUSTIC WASH (TIME ONLY)', [3].STEPS[4].TYPE := 300, [3].STEPS[4].TIME_SPT := 30.0, [3].STEPS[4].REF_FILE := 2164745, [3].STEPS[5].NAME := 'CAUSTIC TO DRAIN', [3].STEPS[5].TYPE := 100, [3].STEPS[5].TIME_SPT := 0.5, [3].STEPS[5].REF_FILE := 2164745, [3].STEPS[6].NAME := 'POST RINSE', [3].STEPS[6].TYPE := 100, [3].STEPS[6].TIME_SPT := 5.0, [3].STEPS[6].REF_FILE := 2164745, [3].STEPS[7].NAME := 'SANITIZE', [3].STEPS[7].TYPE := 600, [3].STEPS[7].TIME_SPT := 5.0,
        [3].STEPS[7].REF_FILE := 2164745, [3].STEPS[8].NAME := 'SANITIZE TO DRAIN', [3].STEPS[8].TYPE := 100, [3].STEPS[8].TIME_SPT := 5.0, [3].STEPS[8].REF_FILE := 2164745, [3].STEPS[9].NAME := 'FINAL RINSE', [3].STEPS[9].TYPE := 100, [3].STEPS[9].TIME_SPT := 5.0, [3].STEPS[9].REF_FILE := 2164745, [3].STEPS[10].NAME := 'FINAL RINSE TO DRAIN', [3].STEPS[10].TYPE := 100, [3].STEPS[10].TIME_SPT := 0.5, [3].STEPS[10].REF_FILE := 2164745, [3].STEPS[11].TYPE := 999, [3].STEPS[12].TYPE := 999, [3].STEPS[13].TYPE := 999, [3].STEPS[14].TYPE := 999, [3].STEPS[15].TYPE := 999, [3].STEPS[16].TYPE := 999, [3].STEPS[17].TYPE := 999, [3].STEPS[18].TYPE := 999, [3].STEPS[19].TYPE := 999, [3].STEPS[20].TYPE := 999, [3].STEPS[21].TYPE := 999, [3].STEPS[22].TYPE := 999, [3].STEPS[23].TYPE := 999, [3].STEPS[24].TYPE := 999, [3].STEPS[25].TYPE := 999, [3].STEPS[26].TYPE := 999, [3].STEPS[27].TYPE := 999, [3].STEPS[28].TYPE := 999, [3].STEPS[29].TYPE := 999, [3].STEPS[30].TYPE := 999, [3].STEPS[31].TYPE := 999, [3].STEPS[32].TYPE := 999, [3].STEPS[33].TYPE := 999, [3].STEPS[34].TYPE := 999, [3].STEPS[35].TYPE := 999, [3].STEPS[36].TYPE := 999, [3].STEPS[37].TYPE := 999, [3].STEPS[38].TYPE := 999, [3].STEPS[39].TYPE := 999, [3].STEPS[40].TYPE := 999, [3].STEPS[41].TYPE := 999, [3].STEPS[42].TYPE := 999, [3].STEPS[43].TYPE := 999, [3].STEPS[44].TYPE := 999, [3].STEPS[45].TYPE := 999, [3].STEPS[46].TYPE := 999, [3].STEPS[47].TYPE := 999, [3].STEPS[48].TYPE := 999, [3].STEPS[49].TYPE := 999, [4].NAME := 'Filler Line Wash', [4].NUMBER := 4, [4].STEPS[0].NAME := 'SYSTEM IDLE', [4].STEPS[1].NAME := 'OPERATOR ACKNOWLEDGE', [4].STEPS[1].TYPE := 50, [4].STEPS[1].REF_FILE := 67379200, [4].STEPS[2].NAME := 'PRERINSE', [4].STEPS[2].TYPE := 100,
        [4].STEPS[2].TIME_SPT := 5.0, [4].STEPS[2].REF_FILE := -2071715837, [4].STEPS[3].NAME := 'PRERINSE TO DRAIN', [4].STEPS[3].TYPE := 100, [4].STEPS[3].TIME_SPT := 0.5, [4].STEPS[3].REF_FILE := 75767811, [4].STEPS[4].NAME := 'CAUSTIC WASH (TIME ONLY)', [4].STEPS[4].TYPE := 300, [4].STEPS[4].TIME_SPT := 30.0, [4].STEPS[4].REF_FILE := 1149509635, [4].STEPS[5].NAME := 'CAUSTIC TO DRAIN', [4].STEPS[5].TYPE := 100, [4].STEPS[5].TIME_SPT := 0.5, [4].STEPS[5].REF_FILE := 75767811, [4].STEPS[6].NAME := 'POST RINSE', [4].STEPS[6].TYPE := 100, [4].STEPS[6].TIME_SPT := 5.0, [4].STEPS[6].REF_FILE := -2071715837, [4].STEPS[7].NAME := 'SANITIZER', [4].STEPS[7].TYPE := 600, [4].STEPS[7].TIME_SPT := 5.0, [4].STEPS[7].REF_FILE := -2071715837, [4].STEPS[8].NAME := 'SANITIZE TO DRAIN', [4].STEPS[8].TYPE := 100, [4].STEPS[8].TIME_SPT := 5.0, [4].STEPS[8].REF_FILE := 75767811, [4].STEPS[9].NAME := 'FINAL RINSE', [4].STEPS[9].TYPE := 100, [4].STEPS[9].TIME_SPT := 5.0, [4].STEPS[9].REF_FILE := -2071715837, [4].STEPS[10].NAME := 'FINAL RINSE TO DRAIN', [4].STEPS[10].TYPE := 100, [4].STEPS[10].TIME_SPT := 0.5, [4].STEPS[10].REF_FILE := 75767815, [4].STEPS[11].TYPE := 999, [4].STEPS[12].TYPE := 999, [4].STEPS[13].TYPE := 999, [4].STEPS[14].TYPE := 999, [4].STEPS[15].TYPE := 999, [4].STEPS[16].TYPE := 999, [4].STEPS[17].TYPE := 999, [4].STEPS[18].TYPE := 999, [4].STEPS[19].TYPE := 999, [4].STEPS[20].TYPE := 999, [4].STEPS[21].TYPE := 999, [4].STEPS[22].TYPE := 999, [4].STEPS[23].TYPE := 999, [4].STEPS[24].TYPE := 999, [4].STEPS[25].TYPE := 999, [4].STEPS[26].TYPE := 999, [4].STEPS[27].TYPE := 999, [4].STEPS[28].TYPE := 999, [4].STEPS[29].TYPE := 999, [4].STEPS[30].TYPE := 999, [4].STEPS[31].TYPE := 999, [4].STEPS[32].TYPE := 999, [4].STEPS[33].TYPE := 999, [4].STEPS[34].TYPE := 999, [4].STEPS[35].TYPE := 999, [4].STEPS[36].TYPE := 999,
        [4].STEPS[37].TYPE := 999, [4].STEPS[38].TYPE := 999, [4].STEPS[39].TYPE := 999, [4].STEPS[40].TYPE := 999, [4].STEPS[41].TYPE := 999, [4].STEPS[42].TYPE := 999, [4].STEPS[43].TYPE := 999, [4].STEPS[44].TYPE := 999, [4].STEPS[45].TYPE := 999, [4].STEPS[46].TYPE := 999, [4].STEPS[47].TYPE := 999, [4].STEPS[48].TYPE := 999, [4].STEPS[49].TYPE := 999, [5].NUMBER := 5, [5].STEPS[0].NAME := 'NOT IN USE', [5].STEPS[1].TYPE := 999, [5].STEPS[2].TYPE := 999, [5].STEPS[3].TYPE := 999, [5].STEPS[4].TYPE := 999, [5].STEPS[5].TYPE := 999, [5].STEPS[6].TYPE := 999, [5].STEPS[7].TYPE := 999, [5].STEPS[8].TYPE := 999, [5].STEPS[9].TYPE := 999, [5].STEPS[10].TYPE := 999, [5].STEPS[11].TYPE := 999, [5].STEPS[12].TYPE := 999, [5].STEPS[13].TYPE := 999, [5].STEPS[14].TYPE := 999, [5].STEPS[15].TYPE := 999, [5].STEPS[16].TYPE := 999, [5].STEPS[17].TYPE := 999, [5].STEPS[18].TYPE := 999, [5].STEPS[19].TYPE := 999, [5].STEPS[20].TYPE := 999, [5].STEPS[21].TYPE := 999, [5].STEPS[22].TYPE := 999, [5].STEPS[23].TYPE := 999, [5].STEPS[24].TYPE := 999, [5].STEPS[25].TYPE := 999, [5].STEPS[26].TYPE := 999, [5].STEPS[27].TYPE := 999, [5].STEPS[28].TYPE := 999, [5].STEPS[29].TYPE := 999, [5].STEPS[30].TYPE := 999, [5].STEPS[31].TYPE := 999, [5].STEPS[32].TYPE := 999, [5].STEPS[33].TYPE := 999, [5].STEPS[34].TYPE := 999, [5].STEPS[35].TYPE := 999, [5].STEPS[36].TYPE := 999, [5].STEPS[37].TYPE := 999, [5].STEPS[38].TYPE := 999, [5].STEPS[39].TYPE := 999, [5].STEPS[40].TYPE := 999, [5].STEPS[41].TYPE := 999, [5].STEPS[42].TYPE := 999, [5].STEPS[43].TYPE := 999, [5].STEPS[44].TYPE := 999, [5].STEPS[45].TYPE := 999,
        [5].STEPS[46].TYPE := 999, [5].STEPS[47].TYPE := 999, [5].STEPS[48].TYPE := 999, [5].STEPS[49].TYPE := 999, [6].NUMBER := 6, [6].STEPS[0].NAME := 'NOT IN USE', [6].STEPS[1].TYPE := 999, [6].STEPS[2].TYPE := 999, [6].STEPS[3].TYPE := 999, [6].STEPS[4].TYPE := 999, [6].STEPS[5].TYPE := 999, [6].STEPS[6].TYPE := 999, [6].STEPS[7].TYPE := 999, [6].STEPS[8].TYPE := 999, [6].STEPS[9].TYPE := 999, [6].STEPS[10].TYPE := 999, [6].STEPS[11].TYPE := 999, [6].STEPS[12].TYPE := 999, [6].STEPS[13].TYPE := 999, [6].STEPS[14].TYPE := 999, [6].STEPS[15].TYPE := 999, [6].STEPS[16].TYPE := 999, [6].STEPS[17].TYPE := 999, [6].STEPS[18].TYPE := 999, [6].STEPS[19].TYPE := 999, [6].STEPS[20].TYPE := 999, [6].STEPS[21].TYPE := 999, [6].STEPS[22].TYPE := 999, [6].STEPS[23].TYPE := 999, [6].STEPS[24].TYPE := 999, [6].STEPS[25].TYPE := 999, [6].STEPS[26].TYPE := 999, [6].STEPS[27].TYPE := 999, [6].STEPS[28].TYPE := 999, [6].STEPS[29].TYPE := 999, [6].STEPS[30].TYPE := 999, [6].STEPS[31].TYPE := 999, [6].STEPS[32].TYPE := 999, [6].STEPS[33].TYPE := 999, [6].STEPS[34].TYPE := 999, [6].STEPS[35].TYPE := 999, [6].STEPS[36].TYPE := 999, [6].STEPS[37].TYPE := 999, [6].STEPS[38].TYPE := 999, [6].STEPS[39].TYPE := 999, [6].STEPS[40].TYPE := 999, [6].STEPS[41].TYPE := 999, [6].STEPS[42].TYPE := 999, [6].STEPS[43].TYPE := 999, [6].STEPS[44].TYPE := 999, [6].STEPS[45].TYPE := 999, [6].STEPS[46].TYPE := 999, [6].STEPS[47].TYPE := 999, [6].STEPS[48].TYPE := 999, [6].STEPS[49].TYPE := 999, [7].NUMBER := 7, [7].STEPS[0].NAME := 'NOT IN USE', [7].STEPS[1].TYPE := 999, [7].STEPS[2].TYPE := 999, [7].STEPS[3].TYPE := 999,
        [7].STEPS[4].TYPE := 999, [7].STEPS[5].TYPE := 999, [7].STEPS[6].TYPE := 999, [7].STEPS[7].TYPE := 999, [7].STEPS[8].TYPE := 999, [7].STEPS[9].TYPE := 999, [7].STEPS[10].TYPE := 999, [7].STEPS[11].TYPE := 999, [7].STEPS[12].TYPE := 999, [7].STEPS[13].TYPE := 999, [7].STEPS[14].TYPE := 999, [7].STEPS[15].TYPE := 999, [7].STEPS[16].TYPE := 999, [7].STEPS[17].TYPE := 999, [7].STEPS[18].TYPE := 999, [7].STEPS[19].TYPE := 999, [7].STEPS[20].TYPE := 999, [7].STEPS[21].TYPE := 999, [7].STEPS[22].TYPE := 999, [7].STEPS[23].TYPE := 999, [7].STEPS[24].TYPE := 999, [7].STEPS[25].TYPE := 999, [7].STEPS[26].TYPE := 999, [7].STEPS[27].TYPE := 999, [7].STEPS[28].TYPE := 999, [7].STEPS[29].TYPE := 999, [7].STEPS[30].TYPE := 999, [7].STEPS[31].TYPE := 999, [7].STEPS[32].TYPE := 999, [7].STEPS[33].TYPE := 999, [7].STEPS[34].TYPE := 999, [7].STEPS[35].TYPE := 999, [7].STEPS[36].TYPE := 999, [7].STEPS[37].TYPE := 999, [7].STEPS[38].TYPE := 999, [7].STEPS[39].TYPE := 999, [7].STEPS[40].TYPE := 999, [7].STEPS[41].TYPE := 999, [7].STEPS[42].TYPE := 999, [7].STEPS[43].TYPE := 999, [7].STEPS[44].TYPE := 999, [7].STEPS[45].TYPE := 999, [7].STEPS[46].TYPE := 999, [7].STEPS[47].TYPE := 999, [7].STEPS[48].TYPE := 999, [7].STEPS[49].TYPE := 999, [8].NUMBER := 8, [8].STEPS[0].NAME := 'NOT IN USE', [8].STEPS[1].TYPE := 999, [8].STEPS[2].TYPE := 999, [8].STEPS[3].TYPE := 999, [8].STEPS[4].TYPE := 999, [8].STEPS[5].TYPE := 999, [8].STEPS[6].TYPE := 999, [8].STEPS[7].TYPE := 999, [8].STEPS[8].TYPE := 999, [8].STEPS[9].TYPE := 999, [8].STEPS[10].TYPE := 999, [8].STEPS[11].TYPE := 999, [8].STEPS[12].TYPE := 999,
        [8].STEPS[13].TYPE := 999, [8].STEPS[14].TYPE := 999, [8].STEPS[15].TYPE := 999, [8].STEPS[16].TYPE := 999, [8].STEPS[17].TYPE := 999, [8].STEPS[18].TYPE := 999, [8].STEPS[19].TYPE := 999, [8].STEPS[20].TYPE := 999, [8].STEPS[21].TYPE := 999, [8].STEPS[22].TYPE := 999, [8].STEPS[23].TYPE := 999, [8].STEPS[24].TYPE := 999, [8].STEPS[25].TYPE := 999, [8].STEPS[26].TYPE := 999, [8].STEPS[27].TYPE := 999, [8].STEPS[28].TYPE := 999, [8].STEPS[29].TYPE := 999, [8].STEPS[30].TYPE := 999, [8].STEPS[31].TYPE := 999, [8].STEPS[32].TYPE := 999, [8].STEPS[33].TYPE := 999, [8].STEPS[34].TYPE := 999, [8].STEPS[35].TYPE := 999, [8].STEPS[36].TYPE := 999, [8].STEPS[37].TYPE := 999, [8].STEPS[38].TYPE := 999, [8].STEPS[39].TYPE := 999, [8].STEPS[40].TYPE := 999, [8].STEPS[41].TYPE := 999, [8].STEPS[42].TYPE := 999, [8].STEPS[43].TYPE := 999, [8].STEPS[44].TYPE := 999, [8].STEPS[45].TYPE := 999, [8].STEPS[46].TYPE := 999, [8].STEPS[47].TYPE := 999, [8].STEPS[48].TYPE := 999, [8].STEPS[49].TYPE := 999, [9].NUMBER := 9, [9].STEPS[0].NAME := 'NOT IN USE', [9].STEPS[1].TYPE := 999, [9].STEPS[2].TYPE := 999, [9].STEPS[3].TYPE := 999, [9].STEPS[4].TYPE := 999, [9].STEPS[5].TYPE := 999, [9].STEPS[6].TYPE := 999, [9].STEPS[7].TYPE := 999, [9].STEPS[8].TYPE := 999, [9].STEPS[9].TYPE := 999, [9].STEPS[10].TYPE := 999, [9].STEPS[11].TYPE := 999, [9].STEPS[12].TYPE := 999, [9].STEPS[13].TYPE := 999, [9].STEPS[14].TYPE := 999, [9].STEPS[15].TYPE := 999, [9].STEPS[16].TYPE := 999, [9].STEPS[17].TYPE := 999, [9].STEPS[18].TYPE := 999, [9].STEPS[19].TYPE := 999, [9].STEPS[20].TYPE := 999, [9].STEPS[21].TYPE := 999,
        [9].STEPS[22].TYPE := 999, [9].STEPS[23].TYPE := 999, [9].STEPS[24].TYPE := 999, [9].STEPS[25].TYPE := 999, [9].STEPS[26].TYPE := 999, [9].STEPS[27].TYPE := 999, [9].STEPS[28].TYPE := 999, [9].STEPS[29].TYPE := 999, [9].STEPS[30].TYPE := 999, [9].STEPS[31].TYPE := 999, [9].STEPS[32].TYPE := 999, [9].STEPS[33].TYPE := 999, [9].STEPS[34].TYPE := 999, [9].STEPS[35].TYPE := 999, [9].STEPS[36].TYPE := 999, [9].STEPS[37].TYPE := 999, [9].STEPS[38].TYPE := 999, [9].STEPS[39].TYPE := 999, [9].STEPS[40].TYPE := 999, [9].STEPS[41].TYPE := 999, [9].STEPS[42].TYPE := 999, [9].STEPS[43].TYPE := 999, [9].STEPS[44].TYPE := 999, [9].STEPS[45].TYPE := 999, [9].STEPS[46].TYPE := 999, [9].STEPS[47].TYPE := 999, [9].STEPS[48].TYPE := 999, [9].STEPS[49].TYPE := 999, [10].NUMBER := 10, [10].STEPS[0].NAME := 'NOT IN USE', [10].STEPS[1].TYPE := 999, [10].STEPS[2].TYPE := 999, [10].STEPS[3].TYPE := 999, [10].STEPS[4].TYPE := 999, [10].STEPS[5].TYPE := 999, [10].STEPS[6].TYPE := 999, [10].STEPS[7].TYPE := 999, [10].STEPS[8].TYPE := 999, [10].STEPS[9].TYPE := 999, [10].STEPS[10].TYPE := 999, [10].STEPS[11].TYPE := 999, [10].STEPS[12].TYPE := 999, [10].STEPS[13].TYPE := 999, [10].STEPS[14].TYPE := 999, [10].STEPS[15].TYPE := 999, [10].STEPS[16].TYPE := 999, [10].STEPS[17].TYPE := 999, [10].STEPS[18].TYPE := 999, [10].STEPS[19].TYPE := 999, [10].STEPS[20].TYPE := 999, [10].STEPS[21].TYPE := 999, [10].STEPS[22].TYPE := 999, [10].STEPS[23].TYPE := 999, [10].STEPS[24].TYPE := 999, [10].STEPS[25].TYPE := 999, [10].STEPS[26].TYPE := 999, [10].STEPS[27].TYPE := 999, [10].STEPS[28].TYPE := 999, [10].STEPS[29].TYPE := 999, [10].STEPS[30].TYPE := 999,
        [10].STEPS[31].TYPE := 999, [10].STEPS[32].TYPE := 999, [10].STEPS[33].TYPE := 999, [10].STEPS[34].TYPE := 999, [10].STEPS[35].TYPE := 999, [10].STEPS[36].TYPE := 999, [10].STEPS[37].TYPE := 999, [10].STEPS[38].TYPE := 999, [10].STEPS[39].TYPE := 999, [10].STEPS[40].TYPE := 999, [10].STEPS[41].TYPE := 999, [10].STEPS[42].TYPE := 999, [10].STEPS[43].TYPE := 999, [10].STEPS[44].TYPE := 999, [10].STEPS[45].TYPE := 999, [10].STEPS[46].TYPE := 999, [10].STEPS[47].TYPE := 999, [10].STEPS[48].TYPE := 999, [10].STEPS[49].TYPE := 999, [11].NUMBER := 11, [11].STEPS[0].NAME := 'NOT IN USE', [11].STEPS[1].TYPE := 999, [11].STEPS[2].TYPE := 999, [11].STEPS[3].TYPE := 999, [11].STEPS[4].TYPE := 999, [11].STEPS[5].TYPE := 999, [11].STEPS[6].TYPE := 999, [11].STEPS[7].TYPE := 999, [11].STEPS[8].TYPE := 999, [11].STEPS[9].TYPE := 999, [11].STEPS[10].TYPE := 999, [11].STEPS[11].TYPE := 999, [11].STEPS[12].TYPE := 999, [11].STEPS[13].TYPE := 999, [11].STEPS[14].TYPE := 999, [11].STEPS[15].TYPE := 999, [11].STEPS[16].TYPE := 999, [11].STEPS[17].TYPE := 999, [11].STEPS[18].TYPE := 999, [11].STEPS[19].TYPE := 999, [11].STEPS[20].TYPE := 999, [11].STEPS[21].TYPE := 999, [11].STEPS[22].TYPE := 999, [11].STEPS[23].TYPE := 999, [11].STEPS[24].TYPE := 999, [11].STEPS[25].TYPE := 999, [11].STEPS[26].TYPE := 999, [11].STEPS[27].TYPE := 999, [11].STEPS[28].TYPE := 999, [11].STEPS[29].TYPE := 999, [11].STEPS[30].TYPE := 999, [11].STEPS[31].TYPE := 999, [11].STEPS[32].TYPE := 999, [11].STEPS[33].TYPE := 999, [11].STEPS[34].TYPE := 999, [11].STEPS[35].TYPE := 999, [11].STEPS[36].TYPE := 999, [11].STEPS[37].TYPE := 999, [11].STEPS[38].TYPE := 999, [11].STEPS[39].TYPE := 999,
        [11].STEPS[40].TYPE := 999, [11].STEPS[41].TYPE := 999, [11].STEPS[42].TYPE := 999, [11].STEPS[43].TYPE := 999, [11].STEPS[44].TYPE := 999, [11].STEPS[45].TYPE := 999, [11].STEPS[46].TYPE := 999, [11].STEPS[47].TYPE := 999, [11].STEPS[48].TYPE := 999, [11].STEPS[49].TYPE := 999, [12].NUMBER := 12, [12].STEPS[0].NAME := 'NOT IN USE', [12].STEPS[1].TYPE := 999, [12].STEPS[2].TYPE := 999, [12].STEPS[3].TYPE := 999, [12].STEPS[4].TYPE := 999, [12].STEPS[5].TYPE := 999, [12].STEPS[6].TYPE := 999, [12].STEPS[7].TYPE := 999, [12].STEPS[8].TYPE := 999, [12].STEPS[9].TYPE := 999, [12].STEPS[10].TYPE := 999, [12].STEPS[11].TYPE := 999, [12].STEPS[12].TYPE := 999, [12].STEPS[13].TYPE := 999, [12].STEPS[14].TYPE := 999, [12].STEPS[15].TYPE := 999, [12].STEPS[16].TYPE := 999, [12].STEPS[17].TYPE := 999, [12].STEPS[18].TYPE := 999, [12].STEPS[19].TYPE := 999, [12].STEPS[20].TYPE := 999, [12].STEPS[21].TYPE := 999, [12].STEPS[22].TYPE := 999, [12].STEPS[23].TYPE := 999, [12].STEPS[24].TYPE := 999, [12].STEPS[25].TYPE := 999, [12].STEPS[26].TYPE := 999, [12].STEPS[27].TYPE := 999, [12].STEPS[28].TYPE := 999, [12].STEPS[29].TYPE := 999, [12].STEPS[30].TYPE := 999, [12].STEPS[31].TYPE := 999, [12].STEPS[32].TYPE := 999, [12].STEPS[33].TYPE := 999, [12].STEPS[34].TYPE := 999, [12].STEPS[35].TYPE := 999, [12].STEPS[36].TYPE := 999, [12].STEPS[37].TYPE := 999, [12].STEPS[38].TYPE := 999, [12].STEPS[39].TYPE := 999, [12].STEPS[40].TYPE := 999, [12].STEPS[41].TYPE := 999, [12].STEPS[42].TYPE := 999, [12].STEPS[43].TYPE := 999, [12].STEPS[44].TYPE := 999, [12].STEPS[45].TYPE := 999, [12].STEPS[46].TYPE := 999, [12].STEPS[47].TYPE := 999, [12].STEPS[48].TYPE := 999,
        [12].STEPS[49].TYPE := 999, [13].NUMBER := 13, [13].STEPS[0].NAME := 'NOT IN USE', [13].STEPS[1].TYPE := 999, [13].STEPS[2].TYPE := 999, [13].STEPS[3].TYPE := 999, [13].STEPS[4].TYPE := 999, [13].STEPS[5].TYPE := 999, [13].STEPS[6].TYPE := 999, [13].STEPS[7].TYPE := 999, [13].STEPS[8].TYPE := 999, [13].STEPS[9].TYPE := 999, [13].STEPS[10].TYPE := 999, [13].STEPS[11].TYPE := 999, [13].STEPS[12].TYPE := 999, [13].STEPS[13].TYPE := 999, [13].STEPS[14].TYPE := 999, [13].STEPS[15].TYPE := 999, [13].STEPS[16].TYPE := 999, [13].STEPS[17].TYPE := 999, [13].STEPS[18].TYPE := 999, [13].STEPS[19].TYPE := 999, [13].STEPS[20].TYPE := 999, [13].STEPS[21].TYPE := 999, [13].STEPS[22].TYPE := 999, [13].STEPS[23].TYPE := 999, [13].STEPS[24].TYPE := 999, [13].STEPS[25].TYPE := 999, [13].STEPS[26].TYPE := 999, [13].STEPS[27].TYPE := 999, [13].STEPS[28].TYPE := 999, [13].STEPS[29].TYPE := 999, [13].STEPS[30].TYPE := 999, [13].STEPS[31].TYPE := 999, [13].STEPS[32].TYPE := 999, [13].STEPS[33].TYPE := 999, [13].STEPS[34].TYPE := 999, [13].STEPS[35].TYPE := 999, [13].STEPS[36].TYPE := 999, [13].STEPS[37].TYPE := 999, [13].STEPS[38].TYPE := 999, [13].STEPS[39].TYPE := 999, [13].STEPS[40].TYPE := 999, [13].STEPS[41].TYPE := 999, [13].STEPS[42].TYPE := 999, [13].STEPS[43].TYPE := 999, [13].STEPS[44].TYPE := 999, [13].STEPS[45].TYPE := 999, [13].STEPS[46].TYPE := 999, [13].STEPS[47].TYPE := 999, [13].STEPS[48].TYPE := 999, [13].STEPS[49].TYPE := 999, [14].NUMBER := 14, [14].STEPS[0].NAME := 'NOT IN USE', [14].STEPS[1].TYPE := 999, [14].STEPS[2].TYPE := 999, [14].STEPS[3].TYPE := 999, [14].STEPS[4].TYPE := 999, [14].STEPS[5].TYPE := 999, [14].STEPS[6].TYPE := 999,
        [14].STEPS[7].TYPE := 999, [14].STEPS[8].TYPE := 999, [14].STEPS[9].TYPE := 999, [14].STEPS[10].TYPE := 999, [14].STEPS[11].TYPE := 999, [14].STEPS[12].TYPE := 999, [14].STEPS[13].TYPE := 999, [14].STEPS[14].TYPE := 999, [14].STEPS[15].TYPE := 999, [14].STEPS[16].TYPE := 999, [14].STEPS[17].TYPE := 999, [14].STEPS[18].TYPE := 999, [14].STEPS[19].TYPE := 999, [14].STEPS[20].TYPE := 999, [14].STEPS[21].TYPE := 999, [14].STEPS[22].TYPE := 999, [14].STEPS[23].TYPE := 999, [14].STEPS[24].TYPE := 999, [14].STEPS[25].TYPE := 999, [14].STEPS[26].TYPE := 999, [14].STEPS[27].TYPE := 999, [14].STEPS[28].TYPE := 999, [14].STEPS[29].TYPE := 999, [14].STEPS[30].TYPE := 999, [14].STEPS[31].TYPE := 999, [14].STEPS[32].TYPE := 999, [14].STEPS[33].TYPE := 999, [14].STEPS[34].TYPE := 999, [14].STEPS[35].TYPE := 999, [14].STEPS[36].TYPE := 999, [14].STEPS[37].TYPE := 999, [14].STEPS[38].TYPE := 999, [14].STEPS[39].TYPE := 999, [14].STEPS[40].TYPE := 999, [14].STEPS[41].TYPE := 999, [14].STEPS[42].TYPE := 999, [14].STEPS[43].TYPE := 999, [14].STEPS[44].TYPE := 999, [14].STEPS[45].TYPE := 999, [14].STEPS[46].TYPE := 999, [14].STEPS[47].TYPE := 999, [14].STEPS[48].TYPE := 999, [14].STEPS[49].TYPE := 999, [15].NUMBER := 15, [15].STEPS[0].NAME := 'NOT IN USE', [15].STEPS[1].TYPE := 999, [15].STEPS[2].TYPE := 999, [15].STEPS[3].TYPE := 999, [15].STEPS[4].TYPE := 999, [15].STEPS[5].TYPE := 999, [15].STEPS[6].TYPE := 999, [15].STEPS[7].TYPE := 999, [15].STEPS[8].TYPE := 999, [15].STEPS[9].TYPE := 999, [15].STEPS[10].TYPE := 999, [15].STEPS[11].TYPE := 999, [15].STEPS[12].TYPE := 999, [15].STEPS[13].TYPE := 999, [15].STEPS[14].TYPE := 999, [15].STEPS[15].TYPE := 999,
        [15].STEPS[16].TYPE := 999, [15].STEPS[17].TYPE := 999, [15].STEPS[18].TYPE := 999, [15].STEPS[19].TYPE := 999, [15].STEPS[20].TYPE := 999, [15].STEPS[21].TYPE := 999, [15].STEPS[22].TYPE := 999, [15].STEPS[23].TYPE := 999, [15].STEPS[24].TYPE := 999, [15].STEPS[25].TYPE := 999, [15].STEPS[26].TYPE := 999, [15].STEPS[27].TYPE := 999, [15].STEPS[28].TYPE := 999, [15].STEPS[29].TYPE := 999, [15].STEPS[30].TYPE := 999, [15].STEPS[31].TYPE := 999, [15].STEPS[32].TYPE := 999, [15].STEPS[33].TYPE := 999, [15].STEPS[34].TYPE := 999, [15].STEPS[35].TYPE := 999, [15].STEPS[36].TYPE := 999, [15].STEPS[37].TYPE := 999, [15].STEPS[38].TYPE := 999, [15].STEPS[39].TYPE := 999, [15].STEPS[40].TYPE := 999, [15].STEPS[41].TYPE := 999, [15].STEPS[42].TYPE := 999, [15].STEPS[43].TYPE := 999, [15].STEPS[44].TYPE := 999, [15].STEPS[45].TYPE := 999, [15].STEPS[46].TYPE := 999, [15].STEPS[47].TYPE := 999, [15].STEPS[48].TYPE := 999, [15].STEPS[49].TYPE := 999, [16].NUMBER := 16, [16].STEPS[0].NAME := 'NOT IN USE', [16].STEPS[1].TYPE := 999, [16].STEPS[2].TYPE := 999, [16].STEPS[3].TYPE := 999, [16].STEPS[4].TYPE := 999, [16].STEPS[5].TYPE := 999, [16].STEPS[6].TYPE := 999, [16].STEPS[7].TYPE := 999, [16].STEPS[8].TYPE := 999, [16].STEPS[9].TYPE := 999, [16].STEPS[10].TYPE := 999, [16].STEPS[11].TYPE := 999, [16].STEPS[12].TYPE := 999, [16].STEPS[13].TYPE := 999, [16].STEPS[14].TYPE := 999, [16].STEPS[15].TYPE := 999, [16].STEPS[16].TYPE := 999, [16].STEPS[17].TYPE := 999, [16].STEPS[18].TYPE := 999, [16].STEPS[19].TYPE := 999, [16].STEPS[20].TYPE := 999, [16].STEPS[21].TYPE := 999, [16].STEPS[22].TYPE := 999, [16].STEPS[23].TYPE := 999, [16].STEPS[24].TYPE := 999,
        [16].STEPS[25].TYPE := 999, [16].STEPS[26].TYPE := 999, [16].STEPS[27].TYPE := 999, [16].STEPS[28].TYPE := 999, [16].STEPS[29].TYPE := 999, [16].STEPS[30].TYPE := 999, [16].STEPS[31].TYPE := 999, [16].STEPS[32].TYPE := 999, [16].STEPS[33].TYPE := 999, [16].STEPS[34].TYPE := 999, [16].STEPS[35].TYPE := 999, [16].STEPS[36].TYPE := 999, [16].STEPS[37].TYPE := 999, [16].STEPS[38].TYPE := 999, [16].STEPS[39].TYPE := 999, [16].STEPS[40].TYPE := 999, [16].STEPS[41].TYPE := 999, [16].STEPS[42].TYPE := 999, [16].STEPS[43].TYPE := 999, [16].STEPS[44].TYPE := 999, [16].STEPS[45].TYPE := 999, [16].STEPS[46].TYPE := 999, [16].STEPS[47].TYPE := 999, [16].STEPS[48].TYPE := 999, [16].STEPS[49].TYPE := 999, [17].NUMBER := 17, [17].STEPS[0].NAME := 'NOT IN USE', [17].STEPS[1].TYPE := 999, [17].STEPS[2].TYPE := 999, [17].STEPS[3].TYPE := 999, [17].STEPS[4].TYPE := 999, [17].STEPS[5].TYPE := 999, [17].STEPS[6].TYPE := 999, [17].STEPS[7].TYPE := 999, [17].STEPS[8].TYPE := 999, [17].STEPS[9].TYPE := 999, [17].STEPS[10].TYPE := 999, [17].STEPS[11].TYPE := 999, [17].STEPS[12].TYPE := 999, [17].STEPS[13].TYPE := 999, [17].STEPS[14].TYPE := 999, [17].STEPS[15].TYPE := 999, [17].STEPS[16].TYPE := 999, [17].STEPS[17].TYPE := 999, [17].STEPS[18].TYPE := 999, [17].STEPS[19].TYPE := 999, [17].STEPS[20].TYPE := 999, [17].STEPS[21].TYPE := 999, [17].STEPS[22].TYPE := 999, [17].STEPS[23].TYPE := 999, [17].STEPS[24].TYPE := 999, [17].STEPS[25].TYPE := 999, [17].STEPS[26].TYPE := 999, [17].STEPS[27].TYPE := 999, [17].STEPS[28].TYPE := 999, [17].STEPS[29].TYPE := 999, [17].STEPS[30].TYPE := 999, [17].STEPS[31].TYPE := 999, [17].STEPS[32].TYPE := 999, [17].STEPS[33].TYPE := 999,
        [17].STEPS[34].TYPE := 999, [17].STEPS[35].TYPE := 999, [17].STEPS[36].TYPE := 999, [17].STEPS[37].TYPE := 999, [17].STEPS[38].TYPE := 999, [17].STEPS[39].TYPE := 999, [17].STEPS[40].TYPE := 999, [17].STEPS[41].TYPE := 999, [17].STEPS[42].TYPE := 999, [17].STEPS[43].TYPE := 999, [17].STEPS[44].TYPE := 999, [17].STEPS[45].TYPE := 999, [17].STEPS[46].TYPE := 999, [17].STEPS[47].TYPE := 999, [17].STEPS[48].TYPE := 999, [17].STEPS[49].TYPE := 999, [18].NUMBER := 18, [18].STEPS[0].NAME := 'NOT IN USE', [18].STEPS[1].TYPE := 999, [18].STEPS[2].TYPE := 999, [18].STEPS[3].TYPE := 999, [18].STEPS[4].TYPE := 999, [18].STEPS[5].TYPE := 999, [18].STEPS[6].TYPE := 999, [18].STEPS[7].TYPE := 999, [18].STEPS[8].TYPE := 999, [18].STEPS[9].TYPE := 999, [18].STEPS[10].TYPE := 999, [18].STEPS[11].TYPE := 999, [18].STEPS[12].TYPE := 999, [18].STEPS[13].TYPE := 999, [18].STEPS[14].TYPE := 999, [18].STEPS[15].TYPE := 999, [18].STEPS[16].TYPE := 999, [18].STEPS[17].TYPE := 999, [18].STEPS[18].TYPE := 999, [18].STEPS[19].TYPE := 999, [18].STEPS[20].TYPE := 999, [18].STEPS[21].TYPE := 999, [18].STEPS[22].TYPE := 999, [18].STEPS[23].TYPE := 999, [18].STEPS[24].TYPE := 999, [18].STEPS[25].TYPE := 999, [18].STEPS[26].TYPE := 999, [18].STEPS[27].TYPE := 999, [18].STEPS[28].TYPE := 999, [18].STEPS[29].TYPE := 999, [18].STEPS[30].TYPE := 999, [18].STEPS[31].TYPE := 999, [18].STEPS[32].TYPE := 999, [18].STEPS[33].TYPE := 999, [18].STEPS[34].TYPE := 999, [18].STEPS[35].TYPE := 999, [18].STEPS[36].TYPE := 999, [18].STEPS[37].TYPE := 999, [18].STEPS[38].TYPE := 999, [18].STEPS[39].TYPE := 999, [18].STEPS[40].TYPE := 999, [18].STEPS[41].TYPE := 999, [18].STEPS[42].TYPE := 999,
        [18].STEPS[43].TYPE := 999, [18].STEPS[44].TYPE := 999, [18].STEPS[45].TYPE := 999, [18].STEPS[46].TYPE := 999, [18].STEPS[47].TYPE := 999, [18].STEPS[48].TYPE := 999, [18].STEPS[49].TYPE := 999, [19].NUMBER := 19, [19].STEPS[0].NAME := 'NOT IN USE', [19].STEPS[1].TYPE := 999, [19].STEPS[2].TYPE := 999, [19].STEPS[3].TYPE := 999, [19].STEPS[4].TYPE := 999, [19].STEPS[5].TYPE := 999, [19].STEPS[6].TYPE := 999, [19].STEPS[7].TYPE := 999, [19].STEPS[8].TYPE := 999, [19].STEPS[9].TYPE := 999, [19].STEPS[10].TYPE := 999, [19].STEPS[11].TYPE := 999, [19].STEPS[12].TYPE := 999, [19].STEPS[13].TYPE := 999, [19].STEPS[14].TYPE := 999, [19].STEPS[15].TYPE := 999, [19].STEPS[16].TYPE := 999, [19].STEPS[17].TYPE := 999, [19].STEPS[18].TYPE := 999, [19].STEPS[19].TYPE := 999, [19].STEPS[20].TYPE := 999, [19].STEPS[21].TYPE := 999, [19].STEPS[22].TYPE := 999, [19].STEPS[23].TYPE := 999, [19].STEPS[24].TYPE := 999, [19].STEPS[25].TYPE := 999, [19].STEPS[26].TYPE := 999, [19].STEPS[27].TYPE := 999, [19].STEPS[28].TYPE := 999, [19].STEPS[29].TYPE := 999, [19].STEPS[30].TYPE := 999, [19].STEPS[31].TYPE := 999, [19].STEPS[32].TYPE := 999, [19].STEPS[33].TYPE := 999, [19].STEPS[34].TYPE := 999, [19].STEPS[35].TYPE := 999, [19].STEPS[36].TYPE := 999, [19].STEPS[37].TYPE := 999, [19].STEPS[38].TYPE := 999, [19].STEPS[39].TYPE := 999, [19].STEPS[40].TYPE := 999, [19].STEPS[41].TYPE := 999, [19].STEPS[42].TYPE := 999, [19].STEPS[43].TYPE := 999, [19].STEPS[44].TYPE := 999, [19].STEPS[45].TYPE := 999, [19].STEPS[46].TYPE := 999, [19].STEPS[47].TYPE := 999, [19].STEPS[48].TYPE := 999, [19].STEPS[49].TYPE := 999, [20].NUMBER := 20, [20].STEPS[0].NAME := 'NOT IN USE',
        [20].STEPS[1].TYPE := 999, [20].STEPS[2].TYPE := 999, [20].STEPS[3].TYPE := 999, [20].STEPS[4].TYPE := 999, [20].STEPS[5].TYPE := 999, [20].STEPS[6].TYPE := 999, [20].STEPS[7].TYPE := 999, [20].STEPS[8].TYPE := 999, [20].STEPS[9].TYPE := 999, [20].STEPS[10].TYPE := 999, [20].STEPS[11].TYPE := 999, [20].STEPS[12].TYPE := 999, [20].STEPS[13].TYPE := 999, [20].STEPS[14].TYPE := 999, [20].STEPS[15].TYPE := 999, [20].STEPS[16].TYPE := 999, [20].STEPS[17].TYPE := 999, [20].STEPS[18].TYPE := 999, [20].STEPS[19].TYPE := 999, [20].STEPS[20].TYPE := 999, [20].STEPS[21].TYPE := 999, [20].STEPS[22].TYPE := 999, [20].STEPS[23].TYPE := 999, [20].STEPS[24].TYPE := 999, [20].STEPS[25].TYPE := 999, [20].STEPS[26].TYPE := 999, [20].STEPS[27].TYPE := 999, [20].STEPS[28].TYPE := 999, [20].STEPS[29].TYPE := 999, [20].STEPS[30].TYPE := 999, [20].STEPS[31].TYPE := 999, [20].STEPS[32].TYPE := 999, [20].STEPS[33].TYPE := 999, [20].STEPS[34].TYPE := 999, [20].STEPS[35].TYPE := 999, [20].STEPS[36].TYPE := 999, [20].STEPS[37].TYPE := 999, [20].STEPS[38].TYPE := 999, [20].STEPS[39].TYPE := 999, [20].STEPS[40].TYPE := 999, [20].STEPS[41].TYPE := 999, [20].STEPS[42].TYPE := 999, [20].STEPS[43].TYPE := 999, [20].STEPS[44].TYPE := 999, [20].STEPS[45].TYPE := 999, [20].STEPS[46].TYPE := 999, [20].STEPS[47].TYPE := 999, [20].STEPS[48].TYPE := 999, [20].STEPS[49].TYPE := 999, [21].NUMBER := 21, [21].STEPS[0].NAME := 'NOT IN USE', [21].STEPS[1].TYPE := 999, [21].STEPS[2].TYPE := 999, [21].STEPS[3].TYPE := 999, [21].STEPS[4].TYPE := 999, [21].STEPS[5].TYPE := 999, [21].STEPS[6].TYPE := 999, [21].STEPS[7].TYPE := 999, [21].STEPS[8].TYPE := 999, [21].STEPS[9].TYPE := 999,
        [21].STEPS[10].TYPE := 999, [21].STEPS[11].TYPE := 999, [21].STEPS[12].TYPE := 999, [21].STEPS[13].TYPE := 999, [21].STEPS[14].TYPE := 999, [21].STEPS[15].TYPE := 999, [21].STEPS[16].TYPE := 999, [21].STEPS[17].TYPE := 999, [21].STEPS[18].TYPE := 999, [21].STEPS[19].TYPE := 999, [21].STEPS[20].TYPE := 999, [21].STEPS[21].TYPE := 999, [21].STEPS[22].TYPE := 999, [21].STEPS[23].TYPE := 999, [21].STEPS[24].TYPE := 999, [21].STEPS[25].TYPE := 999, [21].STEPS[26].TYPE := 999, [21].STEPS[27].TYPE := 999, [21].STEPS[28].TYPE := 999, [21].STEPS[29].TYPE := 999, [21].STEPS[30].TYPE := 999, [21].STEPS[31].TYPE := 999, [21].STEPS[32].TYPE := 999, [21].STEPS[33].TYPE := 999, [21].STEPS[34].TYPE := 999, [21].STEPS[35].TYPE := 999, [21].STEPS[36].TYPE := 999, [21].STEPS[37].TYPE := 999, [21].STEPS[38].TYPE := 999, [21].STEPS[39].TYPE := 999, [21].STEPS[40].TYPE := 999, [21].STEPS[41].TYPE := 999, [21].STEPS[42].TYPE := 999, [21].STEPS[43].TYPE := 999, [21].STEPS[44].TYPE := 999, [21].STEPS[45].TYPE := 999, [21].STEPS[46].TYPE := 999, [21].STEPS[47].TYPE := 999, [21].STEPS[48].TYPE := 999, [21].STEPS[49].TYPE := 999, [22].NUMBER := 22, [22].STEPS[0].NAME := 'NOT IN USE', [22].STEPS[1].TYPE := 999, [22].STEPS[2].TYPE := 999, [22].STEPS[3].TYPE := 999, [22].STEPS[4].TYPE := 999, [22].STEPS[5].TYPE := 999, [22].STEPS[6].TYPE := 999, [22].STEPS[7].TYPE := 999, [22].STEPS[8].TYPE := 999, [22].STEPS[9].TYPE := 999, [22].STEPS[10].TYPE := 999, [22].STEPS[11].TYPE := 999, [22].STEPS[12].TYPE := 999, [22].STEPS[13].TYPE := 999, [22].STEPS[14].TYPE := 999, [22].STEPS[15].TYPE := 999, [22].STEPS[16].TYPE := 999, [22].STEPS[17].TYPE := 999, [22].STEPS[18].TYPE := 999,
        [22].STEPS[19].TYPE := 999, [22].STEPS[20].TYPE := 999, [22].STEPS[21].TYPE := 999, [22].STEPS[22].TYPE := 999, [22].STEPS[23].TYPE := 999, [22].STEPS[24].TYPE := 999, [22].STEPS[25].TYPE := 999, [22].STEPS[26].TYPE := 999, [22].STEPS[27].TYPE := 999, [22].STEPS[28].TYPE := 999, [22].STEPS[29].TYPE := 999, [22].STEPS[30].TYPE := 999, [22].STEPS[31].TYPE := 999, [22].STEPS[32].TYPE := 999, [22].STEPS[33].TYPE := 999, [22].STEPS[34].TYPE := 999, [22].STEPS[35].TYPE := 999, [22].STEPS[36].TYPE := 999, [22].STEPS[37].TYPE := 999, [22].STEPS[38].TYPE := 999, [22].STEPS[39].TYPE := 999, [22].STEPS[40].TYPE := 999, [22].STEPS[41].TYPE := 999, [22].STEPS[42].TYPE := 999, [22].STEPS[43].TYPE := 999, [22].STEPS[44].TYPE := 999, [22].STEPS[45].TYPE := 999, [22].STEPS[46].TYPE := 999, [22].STEPS[47].TYPE := 999, [22].STEPS[48].TYPE := 999, [22].STEPS[49].TYPE := 999, [23].NUMBER := 23, [23].STEPS[0].NAME := 'NOT IN USE', [23].STEPS[1].TYPE := 999, [23].STEPS[2].TYPE := 999, [23].STEPS[3].TYPE := 999, [23].STEPS[4].TYPE := 999, [23].STEPS[5].TYPE := 999, [23].STEPS[6].TYPE := 999, [23].STEPS[7].TYPE := 999, [23].STEPS[8].TYPE := 999, [23].STEPS[9].TYPE := 999, [23].STEPS[10].TYPE := 999, [23].STEPS[11].TYPE := 999, [23].STEPS[12].TYPE := 999, [23].STEPS[13].TYPE := 999, [23].STEPS[14].TYPE := 999, [23].STEPS[15].TYPE := 999, [23].STEPS[16].TYPE := 999, [23].STEPS[17].TYPE := 999, [23].STEPS[18].TYPE := 999, [23].STEPS[19].TYPE := 999, [23].STEPS[20].TYPE := 999, [23].STEPS[21].TYPE := 999, [23].STEPS[22].TYPE := 999, [23].STEPS[23].TYPE := 999, [23].STEPS[24].TYPE := 999, [23].STEPS[25].TYPE := 999, [23].STEPS[26].TYPE := 999, [23].STEPS[27].TYPE := 999,
        [23].STEPS[28].TYPE := 999, [23].STEPS[29].TYPE := 999, [23].STEPS[30].TYPE := 999, [23].STEPS[31].TYPE := 999, [23].STEPS[32].TYPE := 999, [23].STEPS[33].TYPE := 999, [23].STEPS[34].TYPE := 999, [23].STEPS[35].TYPE := 999, [23].STEPS[36].TYPE := 999, [23].STEPS[37].TYPE := 999, [23].STEPS[38].TYPE := 999, [23].STEPS[39].TYPE := 999, [23].STEPS[40].TYPE := 999, [23].STEPS[41].TYPE := 999, [23].STEPS[42].TYPE := 999, [23].STEPS[43].TYPE := 999, [23].STEPS[44].TYPE := 999, [23].STEPS[45].TYPE := 999, [23].STEPS[46].TYPE := 999, [23].STEPS[47].TYPE := 999, [23].STEPS[48].TYPE := 999, [23].STEPS[49].TYPE := 999, [24].NUMBER := 24, [24].STEPS[0].NAME := 'NOT IN USE', [24].STEPS[1].TYPE := 999, [24].STEPS[2].TYPE := 999, [24].STEPS[3].TYPE := 999, [24].STEPS[4].TYPE := 999, [24].STEPS[5].TYPE := 999, [24].STEPS[6].TYPE := 999, [24].STEPS[7].TYPE := 999, [24].STEPS[8].TYPE := 999, [24].STEPS[9].TYPE := 999, [24].STEPS[10].TYPE := 999, [24].STEPS[11].TYPE := 999, [24].STEPS[12].TYPE := 999, [24].STEPS[13].TYPE := 999, [24].STEPS[14].TYPE := 999, [24].STEPS[15].TYPE := 999, [24].STEPS[16].TYPE := 999, [24].STEPS[17].TYPE := 999, [24].STEPS[18].TYPE := 999, [24].STEPS[19].TYPE := 999, [24].STEPS[20].TYPE := 999, [24].STEPS[21].TYPE := 999, [24].STEPS[22].TYPE := 999, [24].STEPS[23].TYPE := 999, [24].STEPS[24].TYPE := 999, [24].STEPS[25].TYPE := 999, [24].STEPS[26].TYPE := 999, [24].STEPS[27].TYPE := 999, [24].STEPS[28].TYPE := 999, [24].STEPS[29].TYPE := 999, [24].STEPS[30].TYPE := 999, [24].STEPS[31].TYPE := 999, [24].STEPS[32].TYPE := 999, [24].STEPS[33].TYPE := 999, [24].STEPS[34].TYPE := 999, [24].STEPS[35].TYPE := 999, [24].STEPS[36].TYPE := 999,
        [24].STEPS[37].TYPE := 999, [24].STEPS[38].TYPE := 999, [24].STEPS[39].TYPE := 999, [24].STEPS[40].TYPE := 999, [24].STEPS[41].TYPE := 999, [24].STEPS[42].TYPE := 999, [24].STEPS[43].TYPE := 999, [24].STEPS[44].TYPE := 999, [24].STEPS[45].TYPE := 999, [24].STEPS[46].TYPE := 999, [24].STEPS[47].TYPE := 999, [24].STEPS[48].TYPE := 999, [24].STEPS[49].TYPE := 999, [25].NUMBER := 25, [25].STEPS[0].NAME := 'NOT IN USE', [25].STEPS[1].TYPE := 999, [25].STEPS[2].TYPE := 999, [25].STEPS[3].TYPE := 999, [25].STEPS[4].TYPE := 999, [25].STEPS[5].TYPE := 999, [25].STEPS[6].TYPE := 999, [25].STEPS[7].TYPE := 999, [25].STEPS[8].TYPE := 999, [25].STEPS[9].TYPE := 999, [25].STEPS[10].TYPE := 999, [25].STEPS[11].TYPE := 999, [25].STEPS[12].TYPE := 999, [25].STEPS[13].TYPE := 999, [25].STEPS[14].TYPE := 999, [25].STEPS[15].TYPE := 999, [25].STEPS[16].TYPE := 999, [25].STEPS[17].TYPE := 999, [25].STEPS[18].TYPE := 999, [25].STEPS[19].TYPE := 999, [25].STEPS[20].TYPE := 999, [25].STEPS[21].TYPE := 999, [25].STEPS[22].TYPE := 999, [25].STEPS[23].TYPE := 999, [25].STEPS[24].TYPE := 999, [25].STEPS[25].TYPE := 999, [25].STEPS[26].TYPE := 999, [25].STEPS[27].TYPE := 999, [25].STEPS[28].TYPE := 999, [25].STEPS[29].TYPE := 999, [25].STEPS[30].TYPE := 999, [25].STEPS[31].TYPE := 999, [25].STEPS[32].TYPE := 999, [25].STEPS[33].TYPE := 999, [25].STEPS[34].TYPE := 999, [25].STEPS[35].TYPE := 999, [25].STEPS[36].TYPE := 999, [25].STEPS[37].TYPE := 999, [25].STEPS[38].TYPE := 999, [25].STEPS[39].TYPE := 999, [25].STEPS[40].TYPE := 999, [25].STEPS[41].TYPE := 999, [25].STEPS[42].TYPE := 999, [25].STEPS[43].TYPE := 999, [25].STEPS[44].TYPE := 999, [25].STEPS[45].TYPE := 999,
        [25].STEPS[46].TYPE := 999, [25].STEPS[47].TYPE := 999, [25].STEPS[48].TYPE := 999, [25].STEPS[49].TYPE := 999, [26].NUMBER := 26, [26].STEPS[0].NAME := 'NOT IN USE', [26].STEPS[1].TYPE := 999, [26].STEPS[2].TYPE := 999, [26].STEPS[3].TYPE := 999, [26].STEPS[4].TYPE := 999, [26].STEPS[5].TYPE := 999, [26].STEPS[6].TYPE := 999, [26].STEPS[7].TYPE := 999, [26].STEPS[8].TYPE := 999, [26].STEPS[9].TYPE := 999, [26].STEPS[10].TYPE := 999, [26].STEPS[11].TYPE := 999, [26].STEPS[12].TYPE := 999, [26].STEPS[13].TYPE := 999, [26].STEPS[14].TYPE := 999, [26].STEPS[15].TYPE := 999, [26].STEPS[16].TYPE := 999, [26].STEPS[17].TYPE := 999, [26].STEPS[18].TYPE := 999, [26].STEPS[19].TYPE := 999, [26].STEPS[20].TYPE := 999, [26].STEPS[21].TYPE := 999, [26].STEPS[22].TYPE := 999, [26].STEPS[23].TYPE := 999, [26].STEPS[24].TYPE := 999, [26].STEPS[25].TYPE := 999, [26].STEPS[26].TYPE := 999, [26].STEPS[27].TYPE := 999, [26].STEPS[28].TYPE := 999, [26].STEPS[29].TYPE := 999, [26].STEPS[30].TYPE := 999, [26].STEPS[31].TYPE := 999, [26].STEPS[32].TYPE := 999, [26].STEPS[33].TYPE := 999, [26].STEPS[34].TYPE := 999, [26].STEPS[35].TYPE := 999, [26].STEPS[36].TYPE := 999, [26].STEPS[37].TYPE := 999, [26].STEPS[38].TYPE := 999, [26].STEPS[39].TYPE := 999, [26].STEPS[40].TYPE := 999, [26].STEPS[41].TYPE := 999, [26].STEPS[42].TYPE := 999, [26].STEPS[43].TYPE := 999, [26].STEPS[44].TYPE := 999, [26].STEPS[45].TYPE := 999, [26].STEPS[46].TYPE := 999, [26].STEPS[47].TYPE := 999, [26].STEPS[48].TYPE := 999, [26].STEPS[49].TYPE := 999, [27].NUMBER := 27, [27].STEPS[0].NAME := 'NOT IN USE', [27].STEPS[1].TYPE := 999, [27].STEPS[2].TYPE := 999, [27].STEPS[3].TYPE := 999,
        [27].STEPS[4].TYPE := 999, [27].STEPS[5].TYPE := 999, [27].STEPS[6].TYPE := 999, [27].STEPS[7].TYPE := 999, [27].STEPS[8].TYPE := 999, [27].STEPS[9].TYPE := 999, [27].STEPS[10].TYPE := 999, [27].STEPS[11].TYPE := 999, [27].STEPS[12].TYPE := 999, [27].STEPS[13].TYPE := 999, [27].STEPS[14].TYPE := 999, [27].STEPS[15].TYPE := 999, [27].STEPS[16].TYPE := 999, [27].STEPS[17].TYPE := 999, [27].STEPS[18].TYPE := 999, [27].STEPS[19].TYPE := 999, [27].STEPS[20].TYPE := 999, [27].STEPS[21].TYPE := 999, [27].STEPS[22].TYPE := 999, [27].STEPS[23].TYPE := 999, [27].STEPS[24].TYPE := 999, [27].STEPS[25].TYPE := 999, [27].STEPS[26].TYPE := 999, [27].STEPS[27].TYPE := 999, [27].STEPS[28].TYPE := 999, [27].STEPS[29].TYPE := 999, [27].STEPS[30].TYPE := 999, [27].STEPS[31].TYPE := 999, [27].STEPS[32].TYPE := 999, [27].STEPS[33].TYPE := 999, [27].STEPS[34].TYPE := 999, [27].STEPS[35].TYPE := 999, [27].STEPS[36].TYPE := 999, [27].STEPS[37].TYPE := 999, [27].STEPS[38].TYPE := 999, [27].STEPS[39].TYPE := 999, [27].STEPS[40].TYPE := 999, [27].STEPS[41].TYPE := 999, [27].STEPS[42].TYPE := 999, [27].STEPS[43].TYPE := 999, [27].STEPS[44].TYPE := 999, [27].STEPS[45].TYPE := 999, [27].STEPS[46].TYPE := 999, [27].STEPS[47].TYPE := 999, [27].STEPS[48].TYPE := 999, [27].STEPS[49].TYPE := 999, [28].NUMBER := 28, [28].STEPS[0].NAME := 'NOT IN USE', [28].STEPS[1].TYPE := 999, [28].STEPS[2].TYPE := 999, [28].STEPS[3].TYPE := 999, [28].STEPS[4].TYPE := 999, [28].STEPS[5].TYPE := 999, [28].STEPS[6].TYPE := 999, [28].STEPS[7].TYPE := 999, [28].STEPS[8].TYPE := 999, [28].STEPS[9].TYPE := 999, [28].STEPS[10].TYPE := 999, [28].STEPS[11].TYPE := 999, [28].STEPS[12].TYPE := 999,
        [28].STEPS[13].TYPE := 999, [28].STEPS[14].TYPE := 999, [28].STEPS[15].TYPE := 999, [28].STEPS[16].TYPE := 999, [28].STEPS[17].TYPE := 999, [28].STEPS[18].TYPE := 999, [28].STEPS[19].TYPE := 999, [28].STEPS[20].TYPE := 999, [28].STEPS[21].TYPE := 999, [28].STEPS[22].TYPE := 999, [28].STEPS[23].TYPE := 999, [28].STEPS[24].TYPE := 999, [28].STEPS[25].TYPE := 999, [28].STEPS[26].TYPE := 999, [28].STEPS[27].TYPE := 999, [28].STEPS[28].TYPE := 999, [28].STEPS[29].TYPE := 999, [28].STEPS[30].TYPE := 999, [28].STEPS[31].TYPE := 999, [28].STEPS[32].TYPE := 999, [28].STEPS[33].TYPE := 999, [28].STEPS[34].TYPE := 999, [28].STEPS[35].TYPE := 999, [28].STEPS[36].TYPE := 999, [28].STEPS[37].TYPE := 999, [28].STEPS[38].TYPE := 999, [28].STEPS[39].TYPE := 999, [28].STEPS[40].TYPE := 999, [28].STEPS[41].TYPE := 999, [28].STEPS[42].TYPE := 999, [28].STEPS[43].TYPE := 999, [28].STEPS[44].TYPE := 999, [28].STEPS[45].TYPE := 999, [28].STEPS[46].TYPE := 999, [28].STEPS[47].TYPE := 999, [28].STEPS[48].TYPE := 999, [28].STEPS[49].TYPE := 999, [29].NUMBER := 29, [29].STEPS[0].NAME := 'NOT IN USE', [29].STEPS[1].TYPE := 999, [29].STEPS[2].TYPE := 999, [29].STEPS[3].TYPE := 999, [29].STEPS[4].TYPE := 999, [29].STEPS[5].TYPE := 999, [29].STEPS[6].TYPE := 999, [29].STEPS[7].TYPE := 999, [29].STEPS[8].TYPE := 999, [29].STEPS[9].TYPE := 999, [29].STEPS[10].TYPE := 999, [29].STEPS[11].TYPE := 999, [29].STEPS[12].TYPE := 999, [29].STEPS[13].TYPE := 999, [29].STEPS[14].TYPE := 999, [29].STEPS[15].TYPE := 999, [29].STEPS[16].TYPE := 999, [29].STEPS[17].TYPE := 999, [29].STEPS[18].TYPE := 999, [29].STEPS[19].TYPE := 999, [29].STEPS[20].TYPE := 999, [29].STEPS[21].TYPE := 999,
        [29].STEPS[22].TYPE := 999, [29].STEPS[23].TYPE := 999, [29].STEPS[24].TYPE := 999, [29].STEPS[25].TYPE := 999, [29].STEPS[26].TYPE := 999, [29].STEPS[27].TYPE := 999, [29].STEPS[28].TYPE := 999, [29].STEPS[29].TYPE := 999, [29].STEPS[30].TYPE := 999, [29].STEPS[31].TYPE := 999, [29].STEPS[32].TYPE := 999, [29].STEPS[33].TYPE := 999, [29].STEPS[34].TYPE := 999, [29].STEPS[35].TYPE := 999, [29].STEPS[36].TYPE := 999, [29].STEPS[37].TYPE := 999, [29].STEPS[38].TYPE := 999, [29].STEPS[39].TYPE := 999, [29].STEPS[40].TYPE := 999, [29].STEPS[41].TYPE := 999, [29].STEPS[42].TYPE := 999, [29].STEPS[43].TYPE := 999, [29].STEPS[44].TYPE := 999, [29].STEPS[45].TYPE := 999, [29].STEPS[46].TYPE := 999, [29].STEPS[47].TYPE := 999, [29].STEPS[48].TYPE := 999, [29].STEPS[49].TYPE := 999);
   CIP_1_PROGRAMS_SPANISH : CIP_PROGRAM[20] := ([1].NAME := 'LAVAR ADEREZO TANQUE 1100', [2].NAME := 'LAVAR ADEREZO TANQUE 1200', [3].NAME := 'LAVADO DE LINEA DE PICADOR', [4].NAME := 'LAVADO DE LINEA DE LLENADO');
   CIP_1_RECIPE_SELECTED_HMI : STRING := 'Filler Line Wash';
   CIP_1_RECIPE_SELECTED_SPANISH_HMI : STRING;
   CIP_1_RESET_PB_HMI : BOOL;
   CIP_1_RETURN_HMI : DINT;   // CIP 1 RETURN LOCATION HMI INDICATOR
   CIP_1_RETURN_TO_CAUSTIC : BOOL;   // CIP 1 RETURN TO CAUSTIC TANK DURING CAUSTIC RETURN STEPS
   CIP_1_RETURN_TO_PRERINSE : BOOL;   // CIP 1 RETURN TO PRE-RINSE TANK DURING CAUSTIC RETURN STEPS
   CIP_1_REVERT_RECIPE_EDITS_PB : BOOL;
   CIP_1_RUN_LATCH : BOOL;
   CIP_1_SANITIZE_SEL_PB : BOOL;   // CIP 1 SANITIZE ONLY HMI SELECT PB 0 = FULL CIP CYCLE 1 = SANITIZE ONLY
   CIP_1_SAVE_RECIPE_EDITS_PB : BOOL;
   CIP_1_SECONDS : DINT;   // CIP 1 SECONDS REMAINING IN MINUTE
   CIP_1_SECONDS_REMAINING : DINT;
   CIP_1_SEQ_CTU : COUNTER := (PRE := 29);   // CIP 1 SEQUENCE STEP COUNTER THIS IS THE SEQUENCE STEP CONTROL
   CIP_1_SEQ_ENABLE : DINT;   // CIP 1 SEQUENCER DATA TO BE ENABLED FOR OPERATION DURING CIP
   CIP_1_SEQ_MEMORY_REG : DINT := 5125;
   CIP_1_START_PB_HMI : BOOL;
   CIP_1_STEP_ADV_ACTIVE : BOOL;   // CIP 1 SEQUENCER STEP ADVANCE ACTIVE
   CIP_1_STEP_ADV_MESSAGE : BOOL;
   CIP_1_STEP_ADV_MESSAGE_CTU : COUNTER := (ACC := 1, DN := 1);
   CIP_1_STEP_ADV_MESSAGE_INT : DINT;
   CIP_1_STEP_ADV_MESSAGE_TIMER : TIMER := (PRE := 1000);
   CIP_1_STEP_ADVANCE : BOOL;   // CIP 1 SEQUENCER MANUAL STEP ADVANCE
   CIP_1_STEP_ADVANCE_PB_HMI : BOOL;
   CIP_1_STEP_AVAIL_NAMES : CIP_STEP_DEF[30] := ([0].NAME := 'SYSTEM IDLE', [1].NAME := 'OPERATOR ACKNOWLEDGE', [1].TYPE := 50, [2].NAME := 'FILL TANKS AND PUMP DOWN', [2].TYPE := 400, [3].NAME := 'PRERINSE FILL LINES', [3].TYPE := 100, [4].NAME := 'PRERINSE', [4].TYPE := 100, [5].NAME := 'PRERINSE PUMP DOWN', [5].TYPE := 400, [6].NAME := 'PRERINSE RECIRCULATE', [6].TYPE := 100, [7].NAME := 'PRERINSE TO DRAIN', [7].TYPE := 100, [8].NAME := 'PRERINSE AIR BLOW', [8].TYPE := 100, [9].NAME := 'HOLD FOR CONDUCTIVITY', [9].TYPE := 300, [10].NAME := 'HOLD FOR TEMPERATURE', [10].TYPE := 200, [11].NAME := 'CAUSTIC WASH (TIME ONLY)', [11].TYPE := 300, [12].NAME := 'CAUSTIC PUMP DOWN', [12].TYPE := 400, [13].NAME := 'CAUSTIC TO DRAIN', [13].TYPE := 100, [14].NAME := 'POST RINSE RECOVER CAUSTIC', [14].TYPE := 500, [15].NAME := 'POST RINSE AIR BLOW', [15].TYPE := 100, [16].NAME := 'POST RINSE PUMP DOWN', [16].TYPE := 400, [17].NAME := 'POST RINSE TO DRAIN', [17].TYPE := 100, [18].NAME := 'POST RINSE', [18].TYPE := 100, [19].NAME := 'SANITIZER FILL LINES', [19].TYPE := 600, [20].NAME := 'SANITIZER', [20].TYPE := 600, [21].NAME := 'SANITIZER AIR BLOW', [21].TYPE := 600, [22].NAME := 'SANITIZER PUMP DOWN', [22].TYPE := 600, [23].NAME := 'SANITIZER TO DRAIN', [23].TYPE := 600, [24].NAME := 'PRESSURE RELEASE', [24].TYPE := 100, [25].NAME := 'SPARE', [26].NAME := 'SPARE', [27].NAME := 'SPARE', [28].NAME := 'SPARE', [29].NAME := 'SPARE');
   CIP_1_STEP_COPY : BOOL;
   CIP_1_STEP_DELETE : BOOL;
   CIP_1_STEP_DELETING : BOOL;
   CIP_1_STEP_ID : INT := 1;
   CIP_1_STEP_INSERT_PB : BOOL;   // CIP1 STEP INSERT PB FROM HMI
   CIP_1_STEP_INSERTING : BOOL;   // CIP1 STEP INSERTING IN PROGRESS
   CIP_1_STOP_DURING_RUN : BOOL;   // CIP 1 SEQUENCER STOPPED DURING RUN
   CIP_1_STOP_PB_HMI : BOOL;
   CIP_1_SUPPLY_TEMP_SPT : DINT;   // CIP 1 SUPPLY TEMP SETPOINT
   CIP_1_TANK_TRANS_VIS_TMR : TIMER := (PRE := 20000);   // CIP 1 TANK TRANSFER VISIBILITY TIMER
   CIP_1_TANK_TRANSITION_HMI : BOOL;   // CIP 1 TANK TRANSITION BANNER VISIBLE ON HMI
   CIP_1_TIME_ELAPSED_MIN : DINT;
   CIP_1_TIME_ELAPSED_SEC : DINT;
   CIP_1_TIME_REMAINING : REAL;
   CIP_1_TIME_REMAINING_MINR : DINT;   // TIME REMAINING IN MINUTES TO HMI
   CIP_1_TIME_REMAINING_SECR : DINT;   // TIME REMAINING IN SECONDS TO HMI
   CIP_Cart_Comm_Failed : BOOL;
   CIP_Circuit_1_Visibility : BOOL;
   CIP_Circuit_2_Visibility : BOOL;
   CIP_Circuit_3_Visibility : BOOL;
   CIP_Circuit_4_Visibility : BOOL := 1;
   CIP_Recipe : CIP_Recipe[16] := ([0].Step_Desc[0] := 'Home');
   CIP_RinseStep_PULSE_ENABLE : BOOL;
   CIP_SUPPLY_PUMP_CIP_ENABLE : BOOL;
   CIP_WashStep_PULSE_ENABLE : BOOL;
   CIPEnabled : BOOL;
   CIPNames : STRING[20] := ([1] := 'CIP 1 - DRESSING TANK 1100', [2] := 'CIP 2 - DRESSING TANK 1200', [3] := 'CIP 3 - CHOPPER LINE', [4] := 'CIP 4 - FILLER LINE');
   CIPNames_Spanish : STRING[20] := ([1] := 'CIP 1 - TANQUE DE ADEREZO 1100', [2] := 'CIP 2 - TANQUE DE ADEREZO 1200', [3] := 'CIP 3 - LINEA DE PICADORES', [4] := 'CIP 4 - LINEA DE LLENADO');
   CIPSelected : DINT;
   CIPSelection : DINT;
   CIPSensorInterlocks_OK : BOOL;
   DaylightSavings : Toggle_Bit;
   DTE_TEST : DINT := 2;   // TEST CIP BIT REMOVE WHEN FULL CIP CODE HAS BEEN COMPLETED ==================== Always True Bit
        .0   // TEST CIP BIT REMOVE WHEN FULL CIP CODE HAS BEEN COMPLETED ==================== Always False Bit
   DummyString : STRING[10] := ([1] := 'CIP 1 - TANQUE DE ADEREZO 1100', [2] := 'CIP 2 - TANQUE DE ADEREZO 1200', [3] := 'CIP 3 - LINEA DE PICADORES', [4] := 'CIP 4 - LINEA DE LLENADO');
   DummyString2 : STRING[20] := ([0] := 'Not Used', [1] := 'Descargar 1100', [2] := 'Descargar 1200');
   DummyString3 : STRING[20] := ([1] := 'Llenar Tanque 1100', [2] := 'Llenar Tanque 1200');
   Filler_Call_For_Product : BOOL;
   FINAL_RINSE_DRAIN_LATCH : BOOL;
   FINAL_RINSE_DRAIN_RUN : BOOL;
   FINAL_RINSE_DRAIN_RUN_CLR : BOOL;   // FINAL RINSE JKFF CLEAR BIT
   FINAL_RINSE_DRAIN_RUN_PB : BOOL;
   FINAL_RINSE_FILL_PB_HMI : BOOL;
   FINAL_RINSE_FILL_RUN : BOOL;
   FINAL_RINSE_FILL_RUN_CLR : BOOL;   // FINAL RINSE JKFF CLEAR BIT
   FinalRinse_Fill_Latch : BOOL;   // Final Rinse Tank Fill Latch
   Flow_Detected : BOOL;
   Force_Time_Sync : BOOL;
   FP1000_CIP_Supply_Ind : DINT := 3;
   FP1001 : DINT;   // Flow Plate 1001 Sensor Interlock
   FP1001_CIP_Return_Ind : DINT := 3;
   GlobalAlmAck : BOOL;
   HMI_Alarms_Active : BOOL;
   HMI_Flow : DINT := 4;
   HMI_Global_Alarm_Ack_PB : BOOL;
   HMI_Operator_Ack_REQUEST : BOOL;   // CIP 1 Operator Acknowledge Request Active to Proceed to Next Step
   HMI_Temp : DINT;
   HMIAlarms : DINT[25];   // Alarm Trigger Array
   HMIAlarmsMsg : STRING64[17,32] := ([0,0] := 'P1001 - Drive Faulted', [0,1] := 'P1001 - Drive Failed To Start', [0,2] := 'P1001 - Drive Stopped While Running', [0,3] := 'P1002 - Drive Faulted', [0,4] := 'P1002 - Drive Failed To Start', [0,5] := 'P1002 - Drive Stopped While Running', [0,6] := 'P1003 - Drive Faulted', [0,7] := 'P1003 - Drive Failed To Start', [0,8] := 'P1003 - Drive Stopped While Running', [0,9] := 'P1004 - Drive Faulted', [0,10] := 'P1004 - Drive Failed To Start', [0,11] := 'P1004 - Drive Stopped While Running', [0,12] := 'AG1101 - Drive Faulted', [0,13] := 'AG1101 - Drive Failed To Start', [0,14] := 'AG1101 - Drive Stopped While Running', [0,15] := 'AG1201 - Drive Faulted', [0,16] := 'AG1201 - Drive Failed To Start', [0,17] := 'AG1201 - Drive Stopped While Running', [0,18] := '[A019]', [0,19] := '[A020]', [0,20] := '[A021]', [0,21] := '[A022]', [0,22] := '[A023]', [0,23] := '[A024]', [0,24] := '[A025]', [0,25] := '[A026]', [0,26] := '[A027]', [0,27] := '[A028]', [0,28] := '[A029]', [0,29] := '[A030]', [0,30] := '[A031]', [0,31] := '[A032]', [1,0] := 'Emergency Stop Pushed', [1,1] := 'CIP Cart Communications Fault', [1,2] := 'CIP Circuit #1 Fault - Jumpers Not Correct', [1,3] := 'CIP Circuit #2 Fault - Jumpers Not Correct', [1,4] := 'CIP Circuit #3 Fault - Jumpers Not Correct', [1,5] := 'CIP Circuit #4 Fault - Jumpers Not Correct', [1,6] := 'CIP Circuit #1 Fault - Tank Not Empty', [1,7] := 'CIP Circuit #2 Fault - Tank Not Empty', [1,8] := '[A041]', [1,9] := '[A042]', [1,10] := '[A043]', [1,11] := '[A044]', [1,12] := '[A045]', [1,13] := '[A046]', [1,14] := '[A047]', [1,15] := '[A048]', [1,16] := '[A049]', [1,17] := '[A050]', [1,18] := '[A051]', [1,19] := '[A052]', [1,20] := '[A053]', [1,21] := '[A054]', [1,22] := '[A055]', [1,23] := '[A056]', [1,24] := '[A057]', [1,25] := '[A058]', [1,26] := '[A059]', [1,27] := '[A060]',
        [1,28] := '[A061]', [1,29] := '[A062]', [1,30] := '[A063]', [1,31] := '[A064]', [2,0] := '[A065]', [2,1] := '[A066]', [2,2] := '[A067]', [2,3] := '[A068]', [2,4] := '[A069]', [2,5] := '[A070]', [2,6] := '[A071]', [2,7] := '[A072]', [2,8] := '[A073]', [2,9] := '[A074]', [2,10] := '[A075]', [2,11] := '[A076]', [2,12] := '[A077]', [2,13] := '[A078]', [2,14] := '[A079]', [2,15] := '[A080]', [2,16] := '[A081]', [2,17] := '[A082]', [2,18] := '[A083]', [2,19] := '[A084]', [2,20] := '[A085]', [2,21] := '[A086]', [2,22] := '[A087]', [2,23] := '[A088]', [2,24] := '[A089]', [2,25] := '[A090]', [2,26] := '[A091]', [2,27] := '[A092]', [2,28] := '[A093]', [2,29] := '[A094]', [2,30] := '[A095]', [2,31] := '[A096]', [3,0] := '[A097]', [3,1] := '[A098]', [3,2] := '[A099]', [3,3] := '[A100]', [3,4] := '[A101]', [3,5] := '[A102]', [3,6] := '[A103]', [3,7] := '[A104]', [3,8] := '[A105]', [3,9] := '[A106]', [3,10] := '[A107]', [3,11] := '[A108]', [3,12] := '[A109]', [3,13] := '[A110]', [3,14] := '[A111]', [3,15] := '[A112]', [3,16] := '[A113]', [3,17] := '[A114]', [3,18] := '[A115]', [3,19] := '[A116]', [3,20] := '[A117]', [3,21] := '[A118]', [3,22] := '[A119]', [3,23] := '[A120]',
        [3,24] := '[A121]', [3,25] := '[A122]', [3,26] := '[A123]', [3,27] := '[A124]', [3,28] := '[A125]', [3,29] := '[A126]', [3,30] := '[A127]', [3,31] := '[A128]', [4,0] := '[A129]', [4,1] := '[A130]', [4,2] := '[A131]', [4,3] := '[A132]', [4,4] := '[A133]', [4,5] := '[A134]', [4,6] := '[A135]', [4,7] := '[A136]', [4,8] := '[A137]', [4,9] := '[A138]', [4,10] := '[A139]', [4,11] := '[A140]', [4,12] := '[A141]', [4,13] := '[A142]', [4,14] := '[A143]', [4,15] := '[A144]', [4,16] := '[A145]', [4,17] := '[A146]', [4,18] := '[A147]', [4,19] := '[A148]', [4,20] := '[A149]', [4,21] := '[A150]', [4,22] := '[A151]', [4,23] := '[A152]', [4,24] := '[A153]', [4,25] := '[A154]', [4,26] := '[A155]', [4,27] := '[A156]', [4,28] := '[A157]', [4,29] := '[A158]', [4,30] := '[A159]', [4,31] := '[A160]', [5,0] := '[A161]', [5,1] := '[A162]', [5,2] := '[A163]', [5,3] := '[A164]', [5,4] := '[A165]', [5,5] := '[A166]', [5,6] := '[A167]', [5,7] := '[A168]', [5,8] := '[A169]', [5,9] := '[A170]', [5,10] := '[A171]', [5,11] := '[A172]', [5,12] := '[A173]', [5,13] := '[A174]', [5,14] := '[A175]', [5,15] := '[A176]', [5,16] := '[A177]', [5,17] := '[A178]', [5,18] := '[A179]', [5,19] := '[A180]',
        [5,20] := '[A181]', [5,21] := '[A182]', [5,22] := '[A183]', [5,23] := '[A184]', [5,24] := '[A185]', [5,25] := '[A186]', [5,26] := '[A187]', [5,27] := '[A188]', [5,28] := '[A189]', [5,29] := '[A190]', [5,30] := '[A191]', [5,31] := '[A192]', [6,0] := '[A193]', [6,1] := '[A194]', [6,2] := '[A195]', [6,3] := '[A196]', [6,4] := '[A197]', [6,5] := '[A198]', [6,6] := '[A199]', [6,7] := '[A200]', [6,8] := '[A201]', [6,9] := '[A202]', [6,10] := '[A203]', [6,11] := '[A204]', [6,12] := '[A205]', [6,13] := '[A206]', [6,14] := '[A207]', [6,15] := '[A208]', [6,16] := '[A209]', [6,17] := '[A210]', [6,18] := '[A211]', [6,19] := '[A212]', [6,20] := '[A213]', [6,21] := '[A214]', [6,22] := '[A215]', [6,23] := '[A216]', [6,24] := '[A217]', [6,25] := '[A218]', [6,26] := '[A219]', [6,27] := '[A220]', [6,28] := '[A221]', [6,29] := '[A222]', [6,30] := '[A223]', [6,31] := '[A224]', [7,0] := '[A225]', [7,1] := '[A226]', [7,2] := '[A227]', [7,3] := '[A228]', [7,4] := '[A229]', [7,5] := '[A230]', [7,6] := '[A231]', [7,7] := '[A232]', [7,8] := '[A233]', [7,9] := '[A234]', [7,10] := '[A235]', [7,11] := '[A236]', [7,12] := '[A237]', [7,13] := '[A238]', [7,14] := '[A239]', [7,15] := '[A240]',
        [7,16] := '[A241]', [7,17] := '[A242]', [7,18] := '[A243]', [7,19] := '[A244]', [7,20] := '[A245]', [7,21] := '[A246]', [7,22] := '[A247]', [7,23] := '[A248]', [7,24] := '[A249]', [7,25] := '[A250]', [7,26] := '[A251]', [7,27] := '[A252]', [7,28] := '[A253]', [7,29] := '[A254]', [7,30] := '[A255]', [7,31] := '[A256]', [8,0] := '[A257]', [8,1] := '[A258]', [8,2] := '[A259]', [8,3] := '[A260]', [8,4] := '[A261]', [8,5] := '[A262]', [8,6] := '[A263]', [8,7] := '[A264]', [8,8] := '[A265]', [8,9] := '[A266]', [8,10] := '[A267]', [8,11] := '[A268]', [8,12] := '[A269]', [8,13] := '[A270]', [8,14] := '[A271]', [8,15] := '[A272]', [8,16] := '[A273]', [8,17] := '[A274]', [8,18] := '[A275]', [8,19] := '[A276]', [8,20] := '[A277]', [8,21] := '[A278]', [8,22] := '[A279]', [8,23] := '[A280]', [8,24] := '[A281]', [8,25] := '[A282]', [8,26] := '[A283]', [8,27] := '[A284]', [8,28] := '[A285]', [8,29] := '[A286]', [8,30] := '[A287]', [8,31] := '[A288]', [9,0] := '[A289]', [9,1] := '[A290]', [9,2] := '[A291]', [9,3] := '[A292]', [9,4] := '[A293]', [9,5] := '[A294]', [9,6] := '[A295]', [9,7] := '[A296]', [9,8] := '[A297]', [9,9] := '[A298]', [9,10] := '[A299]', [9,11] := '[A300]',
        [9,12] := '[A301]', [9,13] := '[A302]', [9,14] := '[A303]', [9,15] := '[A304]', [9,16] := '[A305]', [9,17] := '[A306]', [9,18] := '[A307]', [9,19] := '[A308]', [9,20] := '[A309]', [9,21] := '[A310]', [9,22] := '[A311]', [9,23] := '[A312]', [9,24] := '[A313]', [9,25] := '[A314]', [9,26] := '[A315]', [9,27] := '[A316]', [9,28] := '[A317]', [9,29] := '[A318]', [9,30] := '[A319]', [9,31] := '[A320]', [10,0] := '[A321]', [10,1] := '[A322]', [10,2] := '[A323]', [10,3] := '[A324]', [10,4] := '[A325]', [10,5] := '[A326]', [10,6] := '[A327]', [10,7] := '[A328]', [10,8] := '[A329]', [10,9] := '[A330]', [10,10] := '[A331]', [10,11] := '[A332]', [10,12] := '[A333]', [10,13] := '[A334]', [10,14] := '[A335]', [10,15] := '[A336]', [10,16] := '[A337]', [10,17] := '[A338]', [10,18] := '[A339]', [10,19] := '[A340]', [10,20] := '[A341]', [10,21] := '[A342]', [10,22] := '[A343]', [10,23] := '[A344]', [10,24] := '[A345]', [10,25] := '[A346]', [10,26] := '[A347]', [10,27] := '[A348]', [10,28] := '[A349]', [10,29] := '[A350]', [10,30] := '[A351]', [10,31] := '[A352]', [11,0] := '[A353]', [11,1] := '[A354]', [11,2] := '[A355]', [11,3] := '[A356]', [11,4] := '[A357]', [11,5] := '[A358]', [11,6] := '[A359]', [11,7] := '[A360]',
        [11,8] := '[A361]', [11,9] := '[A362]', [11,10] := '[A363]', [11,11] := '[A364]', [11,12] := '[A365]', [11,13] := '[A366]', [11,14] := '[A367]', [11,15] := '[A368]', [11,16] := '[A369]', [11,17] := '[A370]', [11,18] := '[A371]', [11,19] := '[A372]', [11,20] := '[A373]', [11,21] := '[A374]', [11,22] := '[A375]', [11,23] := '[A376]', [11,24] := '[A377]', [11,25] := '[A378]', [11,26] := '[A379]', [11,27] := '[A380]', [11,28] := '[A381]', [11,29] := '[A382]', [11,30] := '[A383]', [11,31] := '[A384]', [12,0] := '[A385]', [12,1] := '[A386]', [12,2] := '[A387]', [12,3] := '[A388]', [12,4] := '[A389]', [12,5] := '[A390]', [12,6] := '[A391]', [12,7] := '[A392]', [12,8] := '[A393]', [12,9] := '[A394]', [12,10] := '[A395]', [12,11] := '[A396]', [12,12] := '[A397]', [12,13] := '[A398]', [12,14] := '[A399]', [12,15] := '[A400]', [12,16] := '[A401]', [12,17] := '[A402]', [12,18] := '[A403]', [12,19] := '[A404]', [12,20] := '[A405]', [12,21] := '[A406]', [12,22] := '[A407]', [12,23] := '[A408]', [12,24] := '[A409]', [12,25] := '[A410]', [12,26] := '[A411]', [12,27] := '[A412]', [12,28] := '[A413]', [12,29] := '[A414]', [12,30] := '[A415]', [12,31] := '[A416]', [13,0] := '[A417]', [13,1] := '[A418]', [13,2] := '[A419]', [13,3] := '[A420]',
        [13,4] := '[A421]', [13,5] := '[A422]', [13,6] := '[A423]', [13,7] := '[A424]', [13,8] := '[A425]', [13,9] := '[A426]', [13,10] := '[A427]', [13,11] := '[A428]', [13,12] := '[A429]', [13,13] := '[A430]', [13,14] := '[A431]', [13,15] := '[A432]', [13,16] := '[A433]', [13,17] := '[A434]', [13,18] := '[A435]', [13,19] := '[A436]', [13,20] := '[A437]', [13,21] := '[A438]', [13,22] := '[A439]', [13,23] := '[A440]', [13,24] := '[A441]', [13,25] := '[A442]', [13,26] := '[A443]', [13,27] := '[A444]', [13,28] := '[A445]', [13,29] := '[A446]', [13,30] := '[A447]', [13,31] := '[A448]', [14,0] := '[A449]', [14,1] := '[A450]', [14,2] := '[A451]', [14,3] := '[A452]', [14,4] := '[A453]', [14,5] := '[A454]', [14,6] := '[A455]', [14,7] := '[A456]', [14,8] := '[A457]', [14,9] := '[A458]', [14,10] := '[A459]', [14,11] := '[A460]', [14,12] := '[A461]', [14,13] := '[A462]', [14,14] := '[A463]', [14,15] := '[A464]', [14,16] := '[A465]', [14,17] := '[A466]', [14,18] := '[A467]', [14,19] := '[A468]', [14,20] := '[A469]', [14,21] := '[A470]', [14,22] := '[A471]', [14,23] := '[A472]', [14,24] := '[A473]', [14,25] := '[A474]', [14,26] := '[A475]', [14,27] := '[A476]', [14,28] := '[A477]', [14,29] := '[A478]', [14,30] := '[A479]', [14,31] := '[A480]',
        [15,0] := '[A481]', [15,1] := '[A482]', [15,2] := '[A483]', [15,3] := '[A484]', [15,4] := '[A485]', [15,5] := '[A486]', [15,6] := '[A487]', [15,7] := '[A488]', [15,8] := '[A489]', [15,9] := '[A490]', [15,10] := '[A491]', [15,11] := '[A492]', [15,12] := '[A493]', [15,13] := '[A494]', [15,14] := '[A495]', [15,15] := '[A496]', [15,16] := '[A497]', [15,17] := '[A498]', [15,18] := '[A499]', [15,19] := '[A500]', [15,20] := '[A501]', [15,21] := '[A502]', [15,22] := '[A503]', [15,23] := '[A504]', [15,24] := '[A505]', [15,25] := '[A506]', [15,26] := '[A507]', [15,27] := '[A508]', [15,28] := '[A509]', [15,29] := '[A510]', [15,30] := '[A511]', [15,31] := '[A512]', [16,0] := '[A513]', [16,1] := '[A514]', [16,2] := '[A515]', [16,3] := '[A516]', [16,4] := '[A517]', [16,5] := '[A518]', [16,6] := '[A519]', [16,7] := '[A520]', [16,8] := '[A521]', [16,9] := '[A522]', [16,10] := '[A523]', [16,11] := '[A524]', [16,12] := '[A525]', [16,13] := '[A526]', [16,14] := '[A527]', [16,15] := '[A528]', [16,16] := '[A529]', [16,17] := '[A530]', [16,18] := '[A531]', [16,19] := '[A532]', [16,20] := '[A533]', [16,21] := '[A534]', [16,22] := '[A535]', [16,23] := '[A536]', [16,24] := '[A537]', [16,25] := '[A538]', [16,26] := '[A539]', [16,27] := '[A540]',
        [16,28] := '[A541]', [16,29] := '[A542]', [16,30] := '[A543]', [16,31] := '[A544]');   // Alarm Descriptions to Match Alarm Trigger Array
   LocalTime : DateTime := (Year := 2022, Month := 9, Day := 15, Hour := 6, Minute := 59, Second := 12, MicroSecond := 468847);
   LT1101 : DTE_SCP_W_LIM := (Input := -0.34490013, Input_Max := 100.0, Scaled_Max := 100.0, Limit_En := 1);   // Tank 1100 Level Transmitter
   LT1201 : DTE_SCP_W_LIM := (Input := 0.5937958, Input_Max := 100.0, Scaled_Max := 100.0, Output := 0.5937958, Limit_En := 1);   // Tank 1200 Level Transmitter
   LT351C : Level_Sensor := (RawInput := 18034.0, SensorPercentLevel := 101.314606, ActualPercentLevel := 101.213394, SensorUpperRange := 100.0, TankOverFlow := 100.1, TankCapacity := 200.0, ProductDensity := 1.0, Scaled_Max := 100.0, Input_Max := 17800.0, LBS := 445.339, KG := 202.00577);   // Raw Receiving CIP Pre-Rinse Tank Level Transmitter
   LT352C : Level_Sensor := (RawInput := 16394.0, SensorPercentLevel := 92.10113, ActualPercentLevel := 92.009125, SensorUpperRange := 100.0, TankOverFlow := 100.1, TankCapacity := 200.0, ProductDensity := 1.0, Scaled_Max := 100.0, Input_Max := 17800.0, LBS := 404.8402, KG := 183.63551);   // Raw Receiving CIP Caustic Tank Level Transmitter
   LT353C : Level_Sensor := (RawInput := 26918.0, SensorPercentLevel := 180.05353, ActualPercentLevel := 86.33936, SensorUpperRange := 48.0, TankOverFlow := 100.1, TankCapacity := 48.0, ProductDensity := 1.0, Scaled_Max := 48.0, Input_Max := 14950.0, LBS := 91.17437, KG := 41.356693);   // Raw Receiving CIP Final Rinse Tank Level Transmitter
   Message_Visibility_1 : DINT;
   OK_TO_PROCEED_PB_HMI : BOOL;
   OK_TO_PROCEED_PB_TIMER : TIMER := (PRE := 1000);
   ONS : DINT[20];   // ONE_SHOT_BIT
   P1001 : DTE_VFD := (INTERLOCK := 1, SPEED_FWD := 75.0, AUTO_SPEED_SETPOINT := 75.0, FORCE_SPEED_SETPOINT := 50.0, ITEMTAG := 1001, MOA_MODE := 1);   // Dressing Tank Fill Pump
   P1001_CIP_Enable : BOOL;
   P1001_ONS : DINT;
   P1001_Start_Request : BOOL;
   P1002 : DTE_VFD := (INTERLOCK := 1, SPEED_FWD := 100.0, AUTO_SPEED_SETPOINT := 100.0, FORCE_SPEED_SETPOINT := 75.0, ITEMTAG := 1002, MOA_MODE := 1);   // Product Filler Fill Pump
   P1002_CIP_ENABLE : BOOL;
   P1002_ONS : DINT := 1;
   P1003 : DTE_VFD := (INTERLOCK := 1, SPEED_FWD := 60.0, AUTO_SPEED_SETPOINT := 60.0, FORCE_SPEED_SETPOINT := 50.0, ITEMTAG := 1003, MOA_MODE := 1);   // CIP Return Pump
   P1003_CIP_ENABLE : BOOL;
   P1003_ONS : DINT;
   P1003_Start_Delay_TMR1 : TIMER := (PRE := 15000);   // CIP Return Pump Active CIP Circuit 1 Start Delay Timer
   P1003_Start_Delay_TMR2 : TIMER := (PRE := 15000);   // CIP Return Pump Active CIP Circuit 2 Start Delay Timer
   P1004 : DTE_VFD := (SPEED_FWD := 54.0, AUTO_SPEED_SETPOINT := 54.0, FORCE_SPEED_SETPOINT := 50.0, ITEMTAG := 1004, MOA_MODE := 1);   // Filler CIP Return Pump
   P1004_ONS : DINT;
   PRE_RINSE_TANK_LEVEL_OFF_PERC : DINT := 100;   // HMI INPUT OF WATER LEVEL OFF IN %
   PRERINSE_DRAIN_LATCH : BOOL;
   PRERINSE_DRAIN_RUN : BOOL;
   PRERINSE_DRAIN_RUN_CLR : BOOL;
   PRERINSE_DRAIN_RUN_PB : BOOL;
   PreRinse_Fill_Latch : BOOL;   // Pre-Rinse Tank Fill Latch
   PRERINSE_FILL_PB_HMI : BOOL;
   PRERINSE_FILL_RUN : BOOL;
   PRERINSE_FILL_RUN_CLR : BOOL;   // PRE-RINSE FILL JKFF CLEAR BIT
   PRERINSE_PREP_LATCH : BOOL;
   PRERINSE_PREP_RUN : BOOL;
   PRERINSE_PREP_RUN_CLR : BOOL;   // Pre-Rinse Prep JKFF Clear Bit
   PRERINSE_PREP_RUN_PB : BOOL;
   PRERINSE_PREP_TEMP_SPT : REAL := 120.0;
   PRERINSE_PREP_TIME_SPT : REAL := 5.0;
   PRERINSE_TIME_REM : DINT;   // PRERINSE TIME REMAINING
   Pulse_DINT : DINT := -809158586;
   Pulse_LINT : LINT := 1663246751049714;
   Pulse_Sync_Bit : TIMER := (PRE := 5000);
   SANITIZE_ENABLE_TRIGGER : BOOL;   // ADVANCE TRIGGER TO NEXT SANITIZE STEP
   SQO_Clear_Timer : TIMER;
   STEP_TIME_MIN : DINT;   // CIP 1 STEP TIMER CONTROLS TIMING PRESET FOR EACH TIMED STEP TO HMI
   STEP_TIME_SEC : DINT;   // CIP 1 STEP TIMER CONTROLS TIMING PRESET FOR EACH TIMED STEP TO HMI
   Sync_Time_Daily : BOOL;
   TEMP_CIP_PROGRAM : CIP_PROGRAM;
   Temp_Hold_Bit_1 : BOOL;
   Temp_Hold_Bit_2 : BOOL;
   TIMERS : TIMER[30] := ([0].PRE := 500, [0].ACC := 496, [0].EN := 1, [0].TT := 1, [1].PRE := 500, [1].ACC := 500, [3].PRE := 600000, [4].PRE := 300000, [5].PRE := 123000, [8].PRE := 999999999, [10].PRE := 2147483647, [10].ACC := 3590292, [11].PRE := 1500, [12].PRE := 1500, [15].PRE := 1500, [17].PRE := 20, [18].PRE := 99999999, [19].PRE := 2500, [20].PRE := 2500, [21].PRE := 2500, [22].PRE := 1500, [23].PRE := 1500, [24].PRE := 1500, [25].ACC := 2, [25].EN := 1, [25].DN := 1, [27].PRE := 60000, [28].PRE := 10000, [28].ACC := 10000, [28].EN := 1, [28].DN := 1, [29].PRE := 60000);
        [10]   // CIP 1 TOTAL TIME ELAPSED TIMER
        [18]   // CIP 1 STEP HOLD TIME ELAPSED TIMER
        [19]   // PRE-RINSE TANK LEVEL DEBOUNCE TMR
        [20]   // CAUSTIC TANK LEVEL DEBOUNCE TMR
        [21]   // FINAL RINSE TANK LEVEL DEBOUNCE TMR
        [28]   // Exhaust Fan Debounce TMR
        [29]   // Exhaust Fan Debounce TMR
        [3]   // CIP 1 CAUSTIC PREP TIMER
        [4]   // CIP 1 PRE-RINSE PREP TIMER
        [5]   // CIP 1 DEVICE PULSE TIMER
        [8]   // CIP 1 STEP TIME ELAPSED TIMER
        [9]   // CIP 1 STEP TIMER CONTROLS TIMING FOR EACH TIMED STEP
   TK1100_LVL_SCP : DTE_SCP_W_LIM := (Input_Max := 100.0, Scaled_Max := 100.0, Limit_En := 1);   // Tank 1100 Level Remote Display
   TK1100_PID : PID := (KP := 2.0, KI := 1.0, MAXO := 100.0, UPD := 0.5);   // Tank 1100 Level Control
   TK1200_LVL_SCP : DTE_SCP_W_LIM := (Input := 0.60884094, Input_Max := 100.0, Scaled_Max := 100.0, Output := 0.60884094, Limit_En := 1);   // Tank 1200 Level Remote Display
   TK1200_PID : PID := (KP := 2.0, KI := 1.0, MAXO := 100.0, UPD := 0.5);   // Tank 1200 Level Control
   Toggle_DST : BOOL;
   TOTALIZER_MIN : DINT := 59;   // CIP 1 TOTALIZER (MIN)
   TOTALIZER_SEC : DINT := 50292;   // CIP 1 TOTALIZER (SEC)
   Transfer_Start_Complete_TMR : TIMER := (PRE := 30000);
   TransferActive_NoFlow_TMR : TIMER := (PRE := 10000000);
   TransferComplete : BOOL;
   TransferDoneBit : BOOL;
   TransferEnabled : BOOL := 1;
   TransferHold : BOOL;
   TransferNames : STRING[20] := ([1] := 'Fill Tank 1100', [2] := 'Fill Tank 1200');
   TransferNames_Spanish : STRING[20] := ([1] := 'Llenar Tanque 1100', [2] := 'Llenar Tanque 1200');
   TransferOk : BOOL;
   TransferONS : DINT[10];
   TransferPaused : BOOL;
   TransferPausePB : BOOL;
   TransferSelected : DINT := 2;
   TransferSelection : DINT := 1;
   TransferSQO : CONTROL;
   TransferSQOTimesArray : REAL[31];
   TransferStandby : BOOL := 1;
   TransferStart_NoFlow_TMR : TIMER;
   TransferStartPB : BOOL;
   TransferStartPBTimer : TIMER := (PRE := 500);
   TransferStartPBVisibility : BOOL := 1;
   TransferStepAdvance : BOOL;
   TransferStopPB : BOOL;
   TransferTimer : TIMER;
   TT370C : Temperature_Transmitter;
   TT371C : Temperature_Transmitter := (RawInput := 8855.0, Input_Max := 30840.0, ScaledMax := 110.0, MeasuredDegC := 31.583982, DegC := 31.583982, DegF := 88.851166);   // Raw Receiving Truck Wash Water Return Temperature Transmitter
   UnloadEnabled : BOOL;
   UnloadNames : STRING[20] := ([0] := 'Not Used', [1] := 'Unload Tank 1100', [2] := 'Unload Tank 1200');
   UnloadNames_Spanish : STRING[20] := ([0] := 'Not Used', [1] := 'Descargar 1100', [2] := 'Descargar 1200');
   UnloadOk : BOOL;
   UnloadSelected : DINT := 2;
   UnloadSelection : DINT := 1;
   UnloadStandby : BOOL;
   UnloadStartPB : BOOL;
   UnloadStartPBTimer : TIMER := (PRE := 500);
   UnloadStartPBVisibility : BOOL;
   UnloadStopPB : BOOL;
   V1001_CIP_ENABLE : BOOL;
   V1002 : DTE_Air_Valve_v2 := (ALM_PRE := 7000, M := 2, Allowed := 1, ITEMTAG := 1002, MOA_Mode := 1);   // CIP Bypass Valve
   V1002_CIP_ENABLE : BOOL;
   V1002_CIP_PULSE : BOOL;
   V1002_Desc : STRING;
   V1002_PIDName : STRING;
   V1003 : DTE_Air_Valve_v2 := (ALM_PRE := 7000, ITEMTAG := 1003, MOA_Mode := 1);   // Filler Valve
   V1003_CIP_ENABLE : BOOL;
   V1003_CIP_PULSE : BOOL;
   V1003_Desc : STRING;
   V1003_PIDName : STRING;
   V1004 : DTE_Air_Valve_v2 := (ALM_PRE := 7000, M := 2, Allowed := 1, ITEMTAG := 1004, MOA_Mode := 1);   // Filler Valve
   V1004_CIP_ENABLE : BOOL;
   V1004_CIP_PULSE : BOOL;
   V1004_Desc : STRING;
   V1004_PIDName : STRING;
   V1005 : DTE_Air_Valve_v2 := (ALM_PRE := 7000, ITEMTAG := 1005, MOA_Mode := 1);   // Filler Valve
   V1005_CIP_ENABLE : BOOL;
   V1005_CIP_PULSE : BOOL;
   V1005_Desc : STRING;
   V1005_PIDName : STRING;
   V1006 : DTE_Air_Valve_v2 := (ALM_PRE := 7000, ITEMTAG := 1006, MOA_Mode := 1);   // Filler Valve
   V1006_CIP_ENABLE : BOOL;
   V1006_CIP_PULSE : BOOL;
   V1006_Desc : STRING;
   V1006_PIDName : STRING;
   V1007 : DTE_Air_Valve_v2 := (TOFF_OUT_ACC := 1, ALM_PRE := 7000, M := 2, Allowed := 1, ITEMTAG := 1007, MOA_Mode := 1);   // Filler Valve
